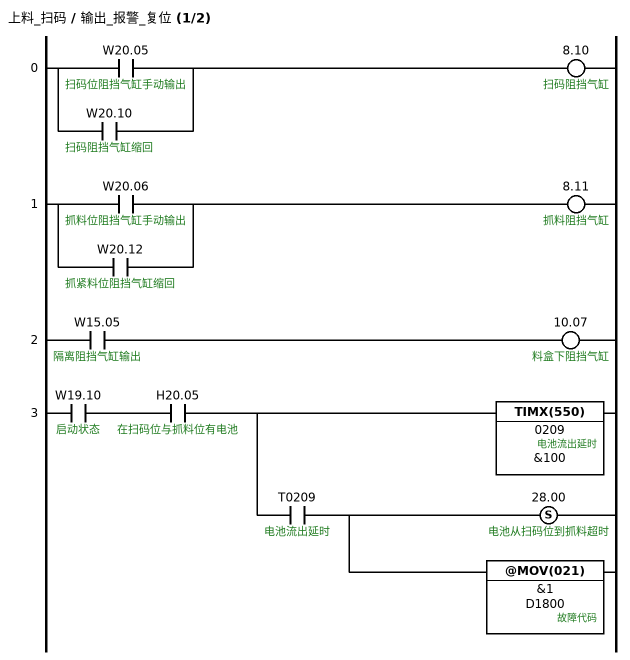
; [picture p72: 上料_扫码 / 输出_报警_复位, rungs 0-3]
; rung 0
LD W20.05  ; 扫码位阻挡气缸手动输出
OR W20.10  ; 扫码阻挡气缸缩回
OUT 8.10  ; 扫码阻挡气缸
; rung 1
LD W20.06  ; 抓料位阻挡气缸手动输出
OR W20.12  ; 抓紧料位阻挡气缸缩回
OUT 8.11  ; 抓料阻挡气缸
; rung 2
LD W15.05  ; 隔离阻挡气缸输出
OUT 10.07  ; 料盒下阻挡气缸
; rung 3
LD W19.10  ; 启动状态
AND H20.05  ; 在扫码位与抓料位有电池
TIMX(550) 0209 &100  ; 电池流出延时
AND T0209  ; 电池流出延时
SET 28.00  ; 电池从扫码位到抓料超时
@MOV(021) &1 D1800  ; 故障代码

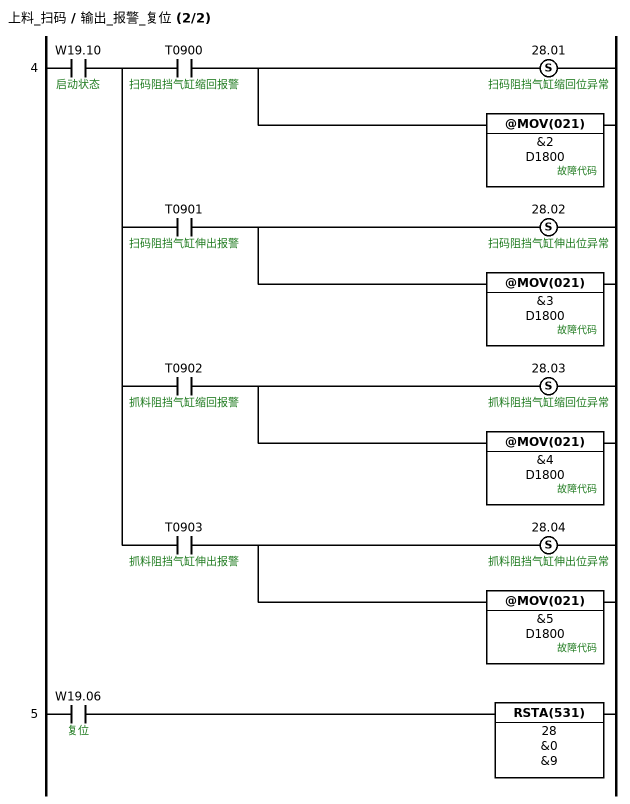
; rung 4
LD W19.10  ; 启动状态
OUT TR0
AND T0900  ; 扫码阻挡气缸缩回报警
SET 28.01  ; 扫码阻挡气缸缩回位异常
@MOV(021) &2 D1800  ; 故障代码
LD TR0
AND T0901  ; 扫码阻挡气缸伸出报警
SET 28.02  ; 扫码阻挡气缸伸出位异常
@MOV(021) &3 D1800  ; 故障代码
LD TR0
AND T0902  ; 抓料阻挡气缸缩回报警
SET 28.03  ; 抓料阻挡气缸缩回位异常
@MOV(021) &4 D1800  ; 故障代码
LD TR0
AND T0903  ; 抓料阻挡气缸伸出报警
SET 28.04  ; 抓料阻挡气缸伸出位异常
@MOV(021) &5 D1800  ; 故障代码
; rung 5
LD W19.06  ; 复位
RSTA(531) 28 &0 &9

### Section END
; rung 0
END(001)

## Program 上料机手 (cyclic task 2)

### Section 上料机械手手动

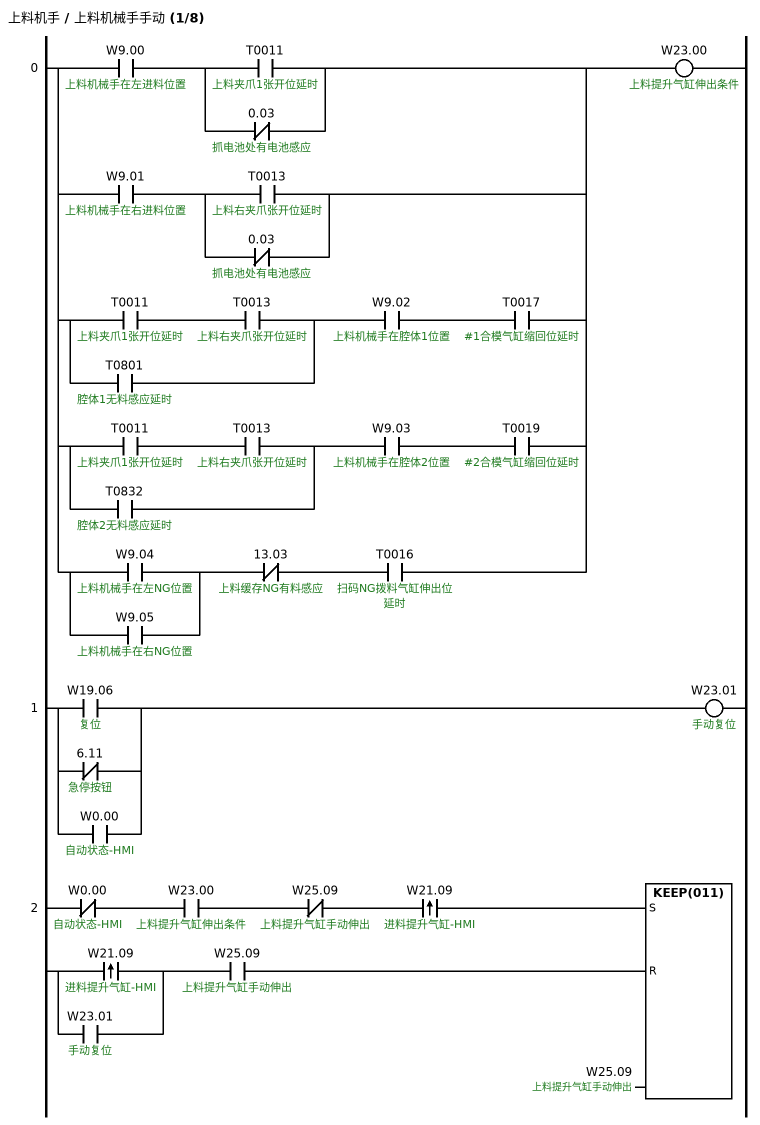
; rung 0
LD W9.00  ; 上料机械手在左进料位置
LD T0011  ; 上料夹爪1张开位延时
ORNOT 0.03  ; 抓电池处有电池感应
ANDLD
LD W9.01  ; 上料机械手在右进料位置
LD T0013  ; 上料右夹爪张开位延时
ORNOT 0.03  ; 抓电池处有电池感应
ANDLD
ORLD
LD T0011  ; 上料夹爪1张开位延时
AND T0013  ; 上料右夹爪张开位延时
OR T0801  ; 腔体1无料感应延时
AND W9.02  ; 上料机械手在腔体1位置
AND T0017  ; #1合模气缸缩回位延时
ORLD
LD T0011  ; 上料夹爪1张开位延时
AND T0013  ; 上料右夹爪张开位延时
OR T0832  ; 腔体2无料感应延时
AND W9.03  ; 上料机械手在腔体2位置
AND T0019  ; #2合模气缸缩回位延时
ORLD
LD W9.04  ; 上料机械手在左NG位置
OR W9.05  ; 上料机械手在右NG位置
ANDNOT 13.03  ; 上料缓存NG有料感应
AND T0016  ; 扫码NG拨料气缸伸出位延时
ORLD
OUT W23.00  ; 上料提升气缸伸出条件
; rung 1
LD W19.06  ; 复位
ORNOT 6.11  ; 急停按钮
OR W0.00  ; 自动状态-HMI
OUT W23.01  ; 手动复位
; rung 2
LDNOT W0.00  ; 自动状态-HMI
AND W23.00  ; 上料提升气缸伸出条件
ANDNOT W25.09  ; 上料提升气缸手动伸出
@AND W21.09  ; 进料提升气缸-HMI
@LD W21.09  ; 进料提升气缸-HMI
OR W23.01  ; 手动复位
AND W25.09  ; 上料提升气缸手动伸出
KEEP(011) W25.09  ; 上料提升气缸手动伸出

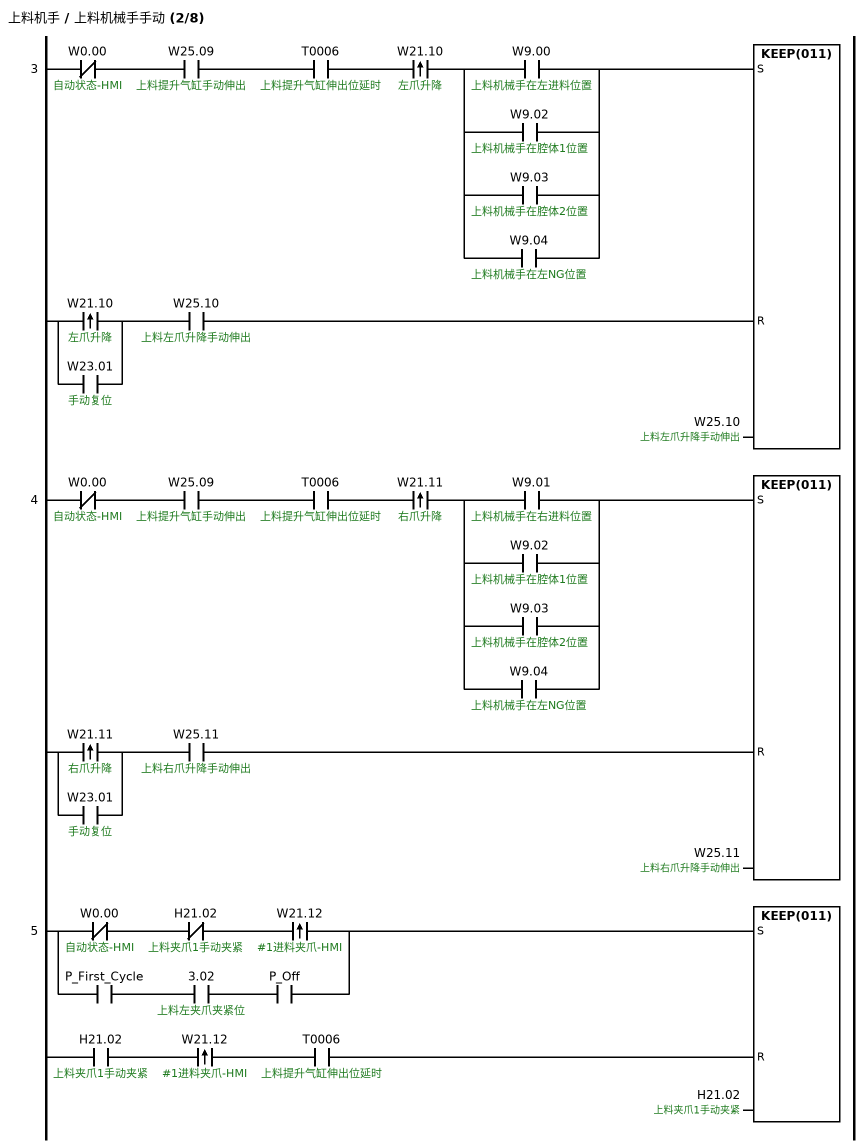
; rung 3
LDNOT W0.00  ; 自动状态-HMI
AND W25.09  ; 上料提升气缸手动伸出
AND T0006  ; 上料提升气缸伸出位延时
@AND W21.10  ; 左爪升降
LD W9.00  ; 上料机械手在左进料位置
OR W9.02  ; 上料机械手在腔体1位置
OR W9.03  ; 上料机械手在腔体2位置
OR W9.04  ; 上料机械手在左NG位置
ANDLD
@LD W21.10  ; 左爪升降
OR W23.01  ; 手动复位
AND W25.10  ; 上料左爪升降手动伸出
KEEP(011) W25.10  ; 上料左爪升降手动伸出
; rung 4
LDNOT W0.00  ; 自动状态-HMI
AND W25.09  ; 上料提升气缸手动伸出
AND T0006  ; 上料提升气缸伸出位延时
@AND W21.11  ; 右爪升降
LD W9.01  ; 上料机械手在右进料位置
OR W9.02  ; 上料机械手在腔体1位置
OR W9.03  ; 上料机械手在腔体2位置
OR W9.04  ; 上料机械手在左NG位置
ANDLD
@LD W21.11  ; 右爪升降
OR W23.01  ; 手动复位
AND W25.11  ; 上料右爪升降手动伸出
KEEP(011) W25.11  ; 上料右爪升降手动伸出
; rung 5
LDNOT W0.00  ; 自动状态-HMI
ANDNOT H21.02  ; 上料夹爪1手动夹紧
@AND W21.12  ; #1进料夹爪-HMI
LD P_First_Cycle
AND 3.02  ; 上料左夹爪夹紧位
AND P_Off
ORLD
LD H21.02  ; 上料夹爪1手动夹紧
@AND W21.12  ; #1进料夹爪-HMI
AND T0006  ; 上料提升气缸伸出位延时
KEEP(011) H21.02  ; 上料夹爪1手动夹紧

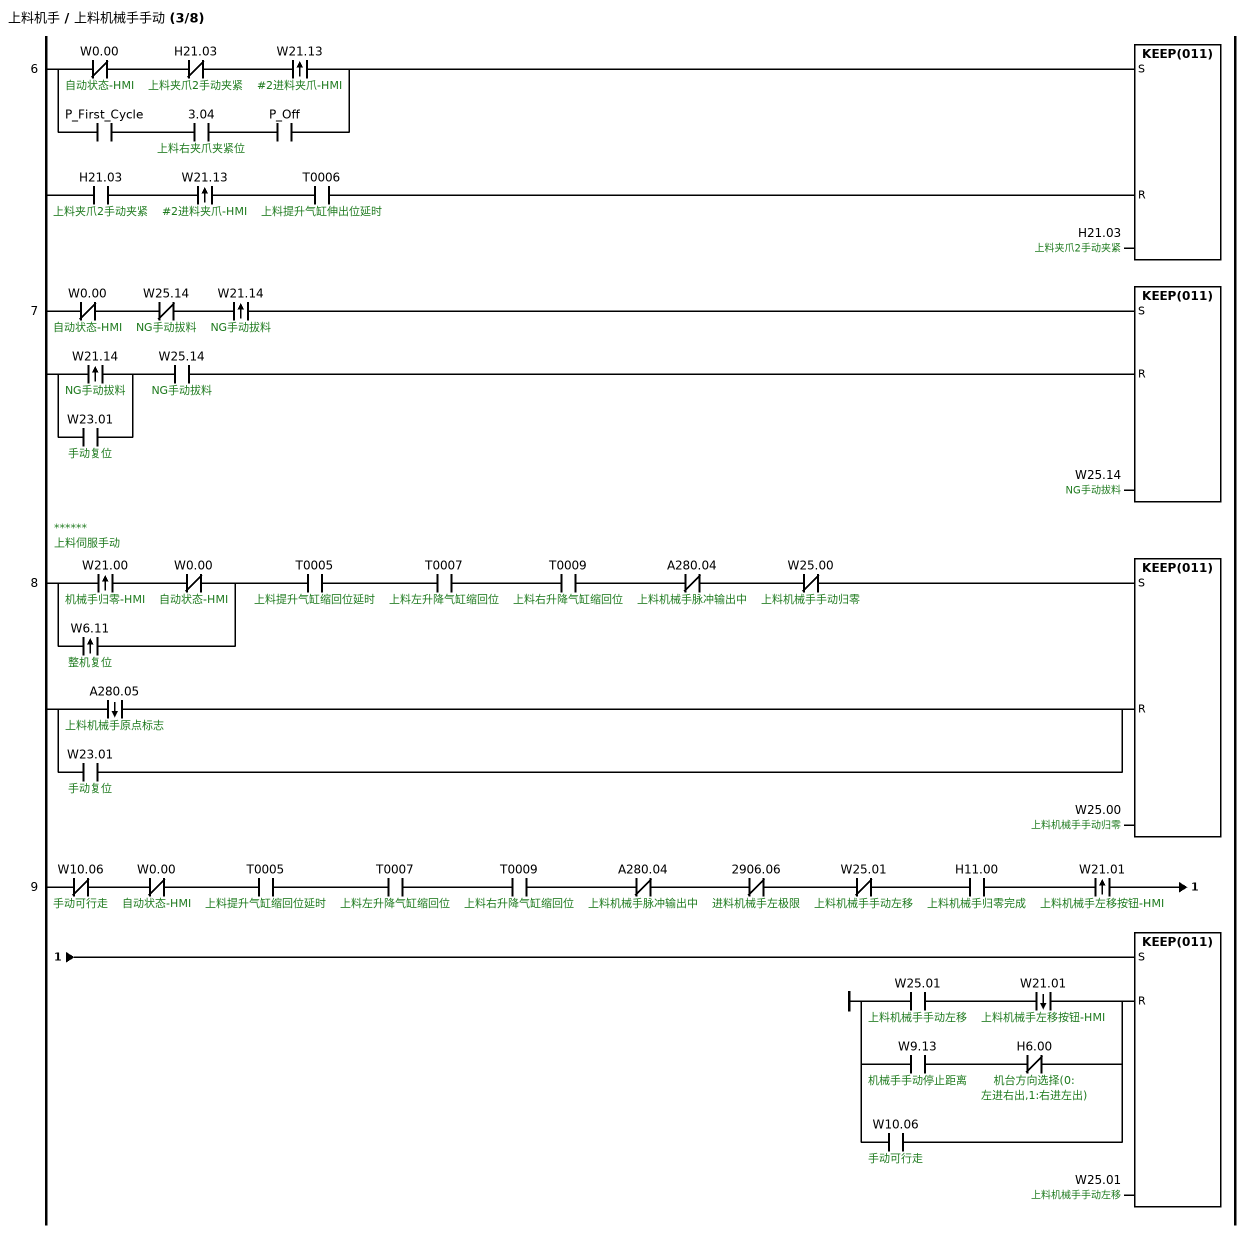
; rung 6
LDNOT W0.00  ; 自动状态-HMI
ANDNOT H21.03  ; 上料夹爪2手动夹紧
@AND W21.13  ; #2进料夹爪-HMI
LD P_First_Cycle
AND 3.04  ; 上料右夹爪夹紧位
AND P_Off
ORLD
LD H21.03  ; 上料夹爪2手动夹紧
@AND W21.13  ; #2进料夹爪-HMI
AND T0006  ; 上料提升气缸伸出位延时
KEEP(011) H21.03  ; 上料夹爪2手动夹紧
; rung 7
LDNOT W0.00  ; 自动状态-HMI
ANDNOT W25.14  ; NG手动拔料
@AND W21.14  ; NG手动拔料
@LD W21.14  ; NG手动拔料
OR W23.01  ; 手动复位
AND W25.14  ; NG手动拔料
KEEP(011) W25.14  ; NG手动拔料
; rung 8: ****** / 上料伺服手动
@LD W21.00  ; 机械手归零-HMI
ANDNOT W0.00  ; 自动状态-HMI
@OR W6.11  ; 整机复位
AND T0005  ; 上料提升气缸缩回位延时
AND T0007  ; 上料左升降气缸缩回位
AND T0009  ; 上料右升降气缸缩回位
ANDNOT A280.04  ; 上料机械手脉冲输出中
ANDNOT W25.00  ; 上料机械手手动归零
%LD A280.05  ; 上料机械手原点标志
OR W23.01  ; 手动复位
KEEP(011) W25.00  ; 上料机械手手动归零
; rung 9
LDNOT W10.06  ; 手动可行走
ANDNOT W0.00  ; 自动状态-HMI
AND T0005  ; 上料提升气缸缩回位延时
AND T0007  ; 上料左升降气缸缩回位
AND T0009  ; 上料右升降气缸缩回位
ANDNOT A280.04  ; 上料机械手脉冲输出中
ANDNOT 2906.06  ; 进料机械手左极限
ANDNOT W25.01  ; 上料机械手手动左移
AND H11.00  ; 上料机械手归零完成
@AND W21.01  ; 上料机械手左移按钮-HMI
LD W25.01  ; 上料机械手手动左移
%AND W21.01  ; 上料机械手左移按钮-HMI
LD W9.13  ; 机械手手动停止距离
ANDNOT H6.00  ; 机台方向选择(0:左进右出,1:右进左出)
ORLD
OR W10.06  ; 手动可行走
KEEP(011) W25.01  ; 上料机械手手动左移

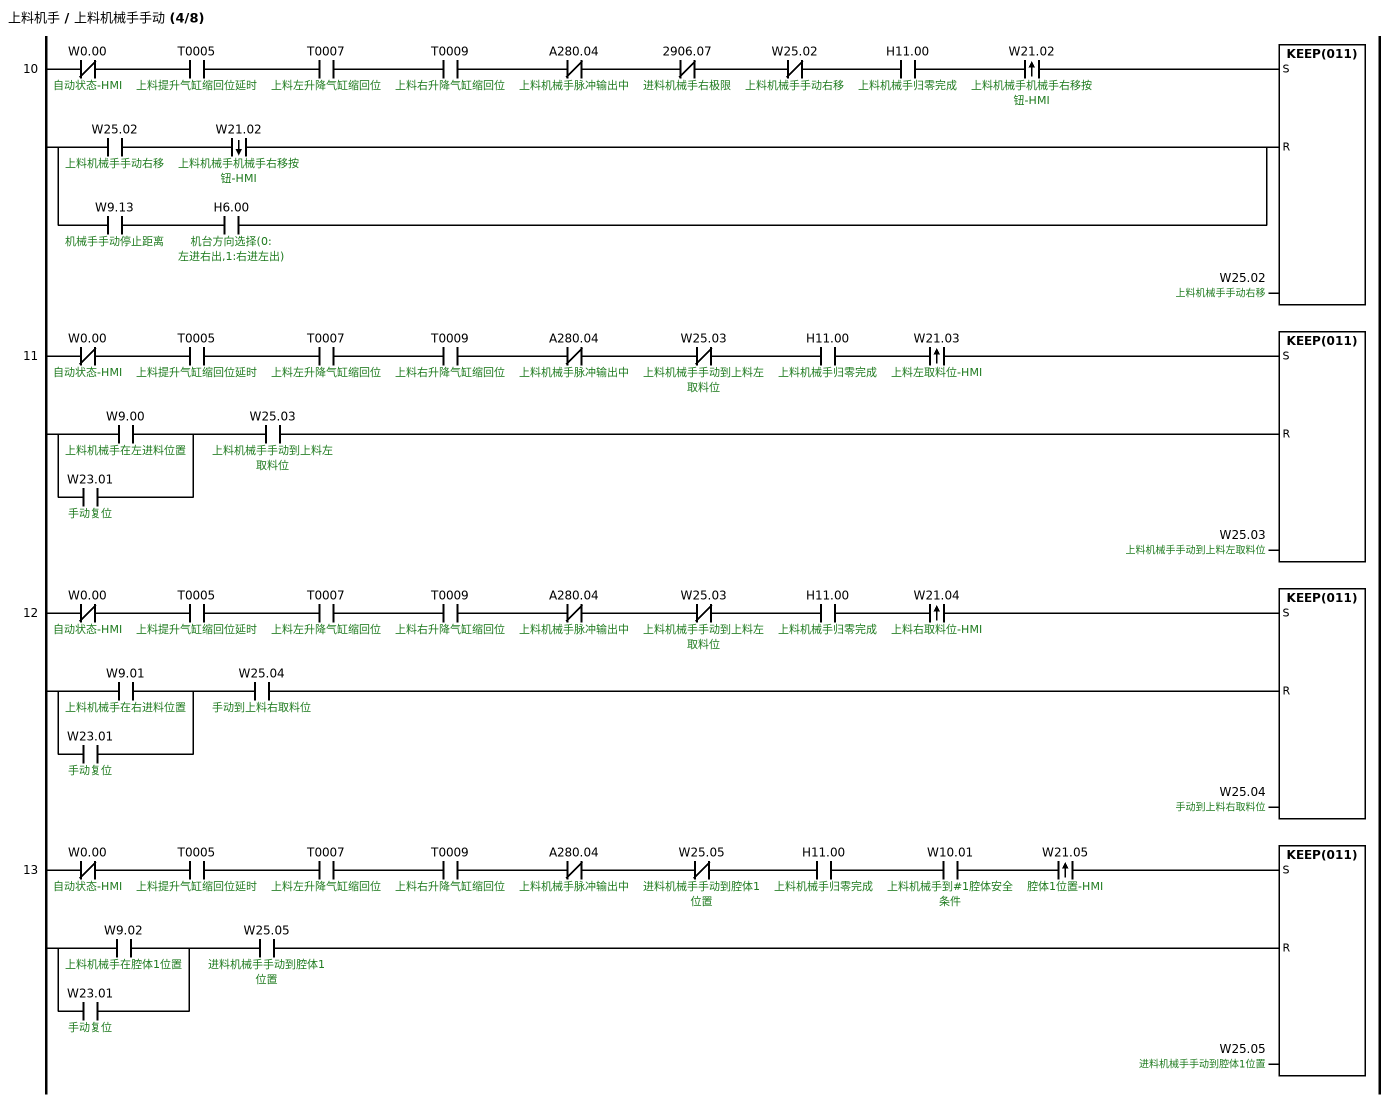
; rung 10
LDNOT W0.00  ; 自动状态-HMI
AND T0005  ; 上料提升气缸缩回位延时
AND T0007  ; 上料左升降气缸缩回位
AND T0009  ; 上料右升降气缸缩回位
ANDNOT A280.04  ; 上料机械手脉冲输出中
ANDNOT 2906.07  ; 进料机械手右极限
ANDNOT W25.02  ; 上料机械手手动右移
AND H11.00  ; 上料机械手归零完成
@AND W21.02  ; 上料机械手机械手右移按钮-HMI
LD W25.02  ; 上料机械手手动右移
%AND W21.02  ; 上料机械手机械手右移按钮-HMI
LD W9.13  ; 机械手手动停止距离
AND H6.00  ; 机台方向选择(0:左进右出,1:右进左出)
ORLD
KEEP(011) W25.02  ; 上料机械手手动右移
; rung 11
LDNOT W0.00  ; 自动状态-HMI
AND T0005  ; 上料提升气缸缩回位延时
AND T0007  ; 上料左升降气缸缩回位
AND T0009  ; 上料右升降气缸缩回位
ANDNOT A280.04  ; 上料机械手脉冲输出中
ANDNOT W25.03  ; 上料机械手手动到上料左取料位
AND H11.00  ; 上料机械手归零完成
@AND W21.03  ; 上料左取料位-HMI
LD W9.00  ; 上料机械手在左进料位置
OR W23.01  ; 手动复位
AND W25.03  ; 上料机械手手动到上料左取料位
KEEP(011) W25.03  ; 上料机械手手动到上料左取料位
; rung 12
LDNOT W0.00  ; 自动状态-HMI
AND T0005  ; 上料提升气缸缩回位延时
AND T0007  ; 上料左升降气缸缩回位
AND T0009  ; 上料右升降气缸缩回位
ANDNOT A280.04  ; 上料机械手脉冲输出中
ANDNOT W25.03  ; 上料机械手手动到上料左取料位
AND H11.00  ; 上料机械手归零完成
@AND W21.04  ; 上料右取料位-HMI
LD W9.01  ; 上料机械手在右进料位置
OR W23.01  ; 手动复位
AND W25.04  ; 手动到上料右取料位
KEEP(011) W25.04  ; 手动到上料右取料位
; rung 13
LDNOT W0.00  ; 自动状态-HMI
AND T0005  ; 上料提升气缸缩回位延时
AND T0007  ; 上料左升降气缸缩回位
AND T0009  ; 上料右升降气缸缩回位
ANDNOT A280.04  ; 上料机械手脉冲输出中
ANDNOT W25.05  ; 进料机械手手动到腔体1位置
AND H11.00  ; 上料机械手归零完成
AND W10.01  ; 上料机械手到#1腔体安全条件
@AND W21.05  ; 腔体1位置-HMI
LD W9.02  ; 上料机械手在腔体1位置
OR W23.01  ; 手动复位
AND W25.05  ; 进料机械手手动到腔体1位置
KEEP(011) W25.05  ; 进料机械手手动到腔体1位置

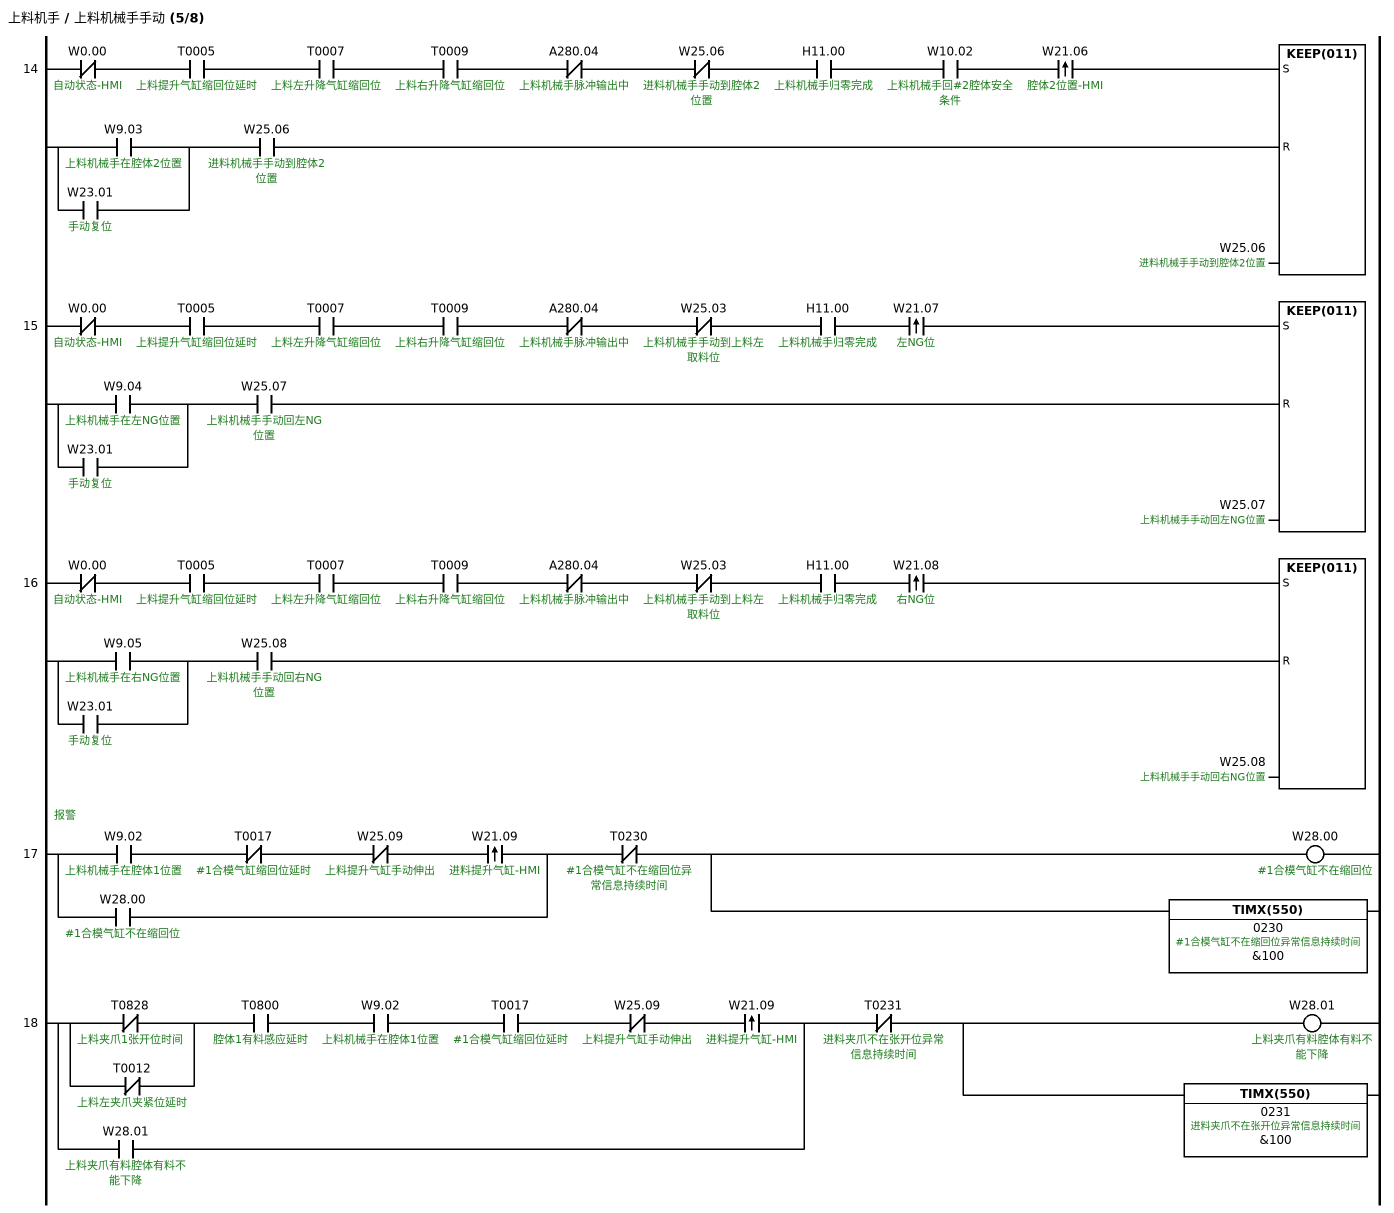
; rung 14
LDNOT W0.00  ; 自动状态-HMI
AND T0005  ; 上料提升气缸缩回位延时
AND T0007  ; 上料左升降气缸缩回位
AND T0009  ; 上料右升降气缸缩回位
ANDNOT A280.04  ; 上料机械手脉冲输出中
ANDNOT W25.06  ; 进料机械手手动到腔体2位置
AND H11.00  ; 上料机械手归零完成
AND W10.02  ; 上料机械手回#2腔体安全条件
@AND W21.06  ; 腔体2位置-HMI
LD W9.03  ; 上料机械手在腔体2位置
OR W23.01  ; 手动复位
AND W25.06  ; 进料机械手手动到腔体2位置
KEEP(011) W25.06  ; 进料机械手手动到腔体2位置
; rung 15
LDNOT W0.00  ; 自动状态-HMI
AND T0005  ; 上料提升气缸缩回位延时
AND T0007  ; 上料左升降气缸缩回位
AND T0009  ; 上料右升降气缸缩回位
ANDNOT A280.04  ; 上料机械手脉冲输出中
ANDNOT W25.03  ; 上料机械手手动到上料左取料位
AND H11.00  ; 上料机械手归零完成
@AND W21.07  ; 左NG位
LD W9.04  ; 上料机械手在左NG位置
OR W23.01  ; 手动复位
AND W25.07  ; 上料机械手手动回左NG位置
KEEP(011) W25.07  ; 上料机械手手动回左NG位置
; rung 16
LDNOT W0.00  ; 自动状态-HMI
AND T0005  ; 上料提升气缸缩回位延时
AND T0007  ; 上料左升降气缸缩回位
AND T0009  ; 上料右升降气缸缩回位
ANDNOT A280.04  ; 上料机械手脉冲输出中
ANDNOT W25.03  ; 上料机械手手动到上料左取料位
AND H11.00  ; 上料机械手归零完成
@AND W21.08  ; 右NG位
LD W9.05  ; 上料机械手在右NG位置
OR W23.01  ; 手动复位
AND W25.08  ; 上料机械手手动回右NG位置
KEEP(011) W25.08  ; 上料机械手手动回右NG位置
; rung 17: 报警
LD W9.02  ; 上料机械手在腔体1位置
ANDNOT T0017  ; #1合模气缸缩回位延时
ANDNOT W25.09  ; 上料提升气缸手动伸出
@AND W21.09  ; 进料提升气缸-HMI
OR W28.00  ; #1合模气缸不在缩回位
ANDNOT T0230  ; #1合模气缸不在缩回位异常信息持续时间
OUT W28.00  ; #1合模气缸不在缩回位
TIMX(550) 0230 &100  ; #1合模气缸不在缩回位异常信息持续时间
; rung 18
LDNOT T0828  ; 上料夹爪1张开位时间
ORNOT T0012  ; 上料左夹爪夹紧位延时
AND T0800  ; 腔体1有料感应延时
AND W9.02  ; 上料机械手在腔体1位置
AND T0017  ; #1合模气缸缩回位延时
ANDNOT W25.09  ; 上料提升气缸手动伸出
@AND W21.09  ; 进料提升气缸-HMI
OR W28.01  ; 上料夹爪有料腔体有料不能下降
ANDNOT T0231  ; 进料夹爪不在张开位异常信息持续时间
OUT W28.01  ; 上料夹爪有料腔体有料不能下降
TIMX(550) 0231 &100  ; 进料夹爪不在张开位异常信息持续时间

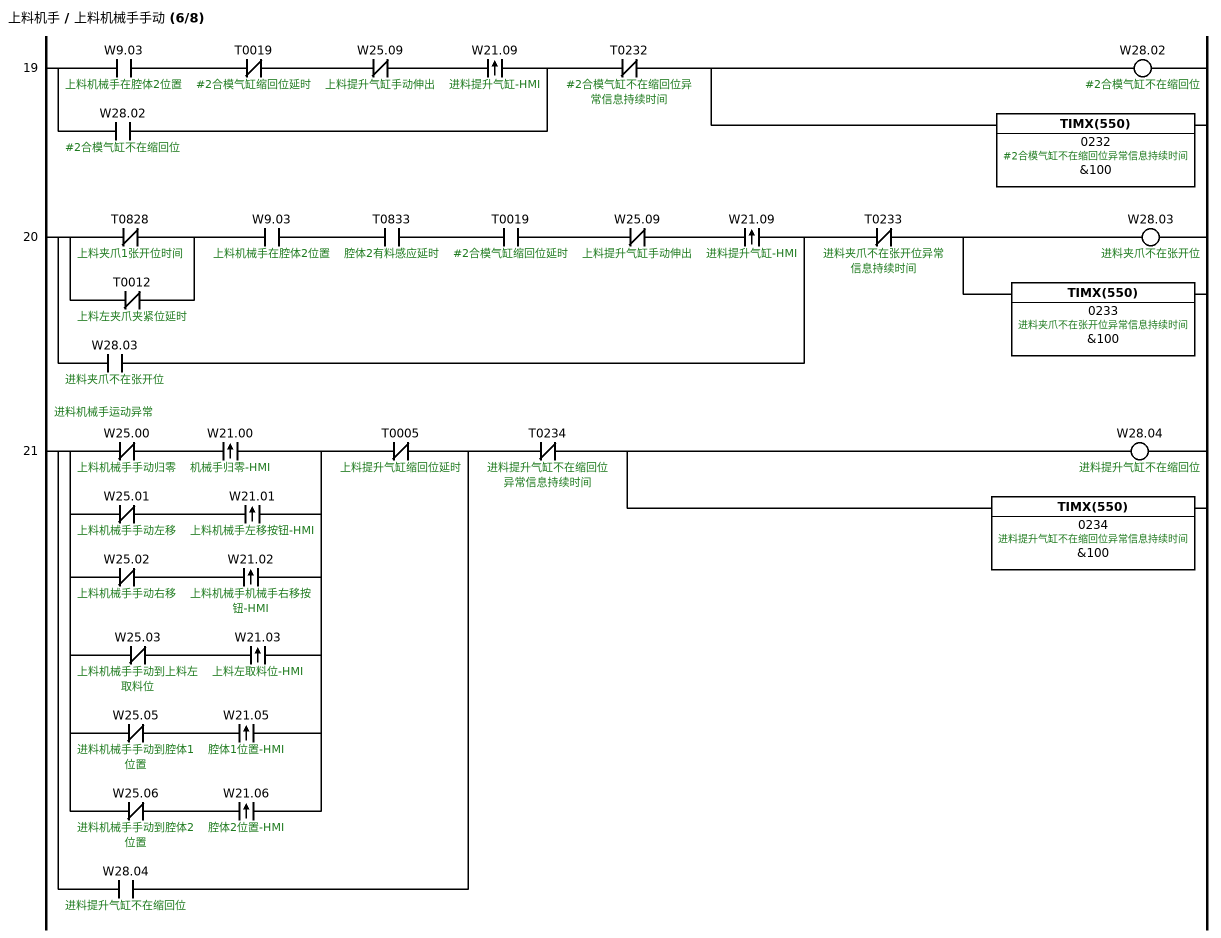
; rung 19
LD W9.03  ; 上料机械手在腔体2位置
ANDNOT T0019  ; #2合模气缸缩回位延时
ANDNOT W25.09  ; 上料提升气缸手动伸出
@AND W21.09  ; 进料提升气缸-HMI
OR W28.02  ; #2合模气缸不在缩回位
ANDNOT T0232  ; #2合模气缸不在缩回位异常信息持续时间
OUT W28.02  ; #2合模气缸不在缩回位
TIMX(550) 0232 &100  ; #2合模气缸不在缩回位异常信息持续时间
; rung 20
LDNOT T0828  ; 上料夹爪1张开位时间
ORNOT T0012  ; 上料左夹爪夹紧位延时
AND W9.03  ; 上料机械手在腔体2位置
AND T0833  ; 腔体2有料感应延时
AND T0019  ; #2合模气缸缩回位延时
ANDNOT W25.09  ; 上料提升气缸手动伸出
@AND W21.09  ; 进料提升气缸-HMI
OR W28.03  ; 进料夹爪不在张开位
ANDNOT T0233  ; 进料夹爪不在张开位异常信息持续时间
OUT W28.03  ; 进料夹爪不在张开位
TIMX(550) 0233 &100  ; 进料夹爪不在张开位异常信息持续时间
; rung 21: 进料机械手运动异常
LDNOT W25.00  ; 上料机械手手动归零
@AND W21.00  ; 机械手归零-HMI
LDNOT W25.01  ; 上料机械手手动左移
@AND W21.01  ; 上料机械手左移按钮-HMI
ORLD
LDNOT W25.02  ; 上料机械手手动右移
@AND W21.02  ; 上料机械手机械手右移按钮-HMI
ORLD
LDNOT W25.03  ; 上料机械手手动到上料左取料位
@AND W21.03  ; 上料左取料位-HMI
ORLD
LDNOT W25.05  ; 进料机械手手动到腔体1位置
@AND W21.05  ; 腔体1位置-HMI
ORLD
LDNOT W25.06  ; 进料机械手手动到腔体2位置
@AND W21.06  ; 腔体2位置-HMI
ORLD
ANDNOT T0005  ; 上料提升气缸缩回位延时
OR W28.04  ; 进料提升气缸不在缩回位
ANDNOT T0234  ; 进料提升气缸不在缩回位异常信息持续时间
OUT W28.04  ; 进料提升气缸不在缩回位
TIMX(550) 0234 &100  ; 进料提升气缸不在缩回位异常信息持续时间

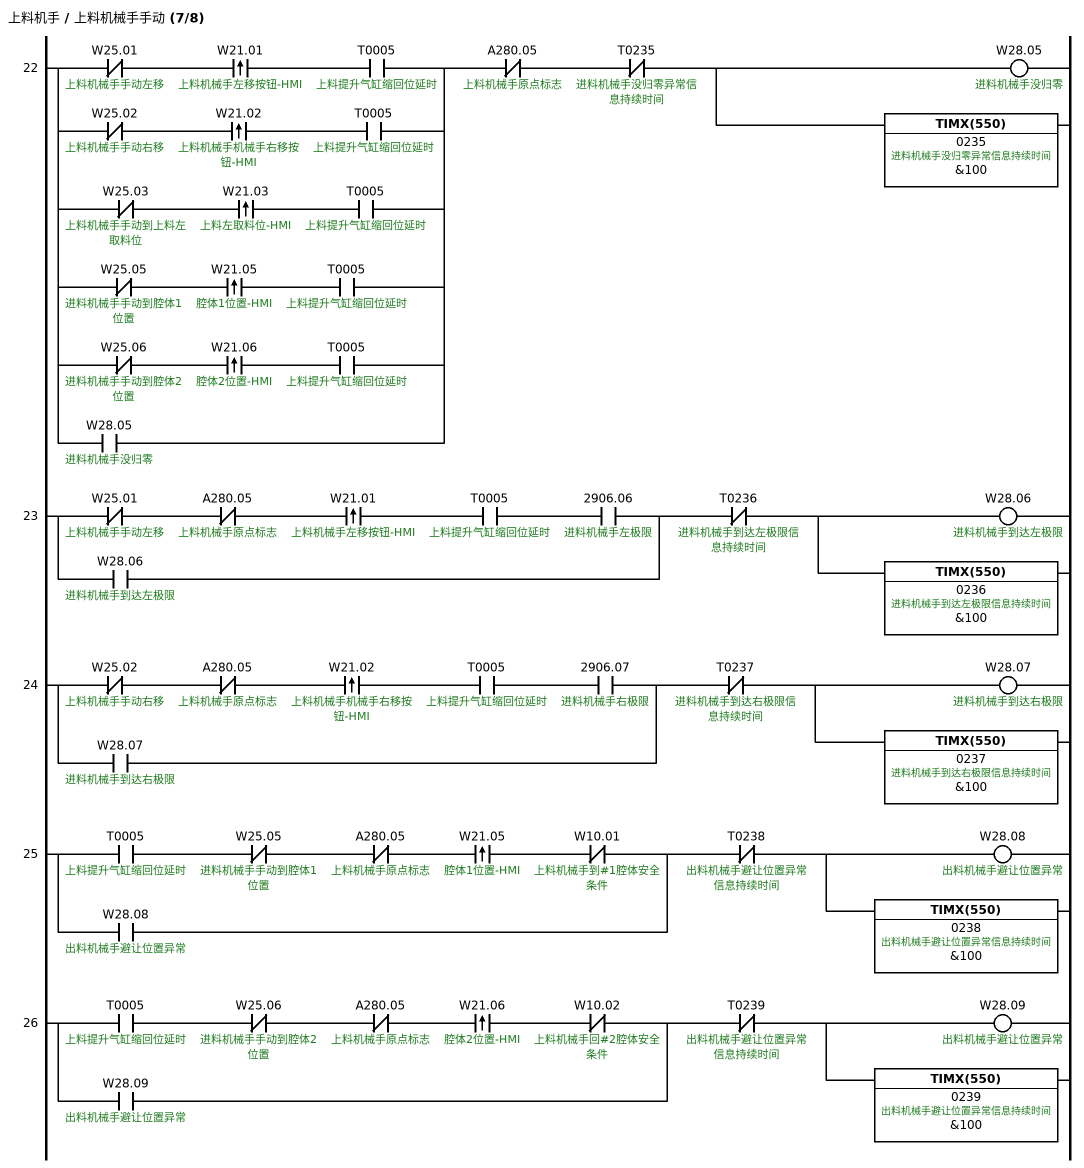
; rung 22
LDNOT W25.01  ; 上料机械手手动左移
@AND W21.01  ; 上料机械手左移按钮-HMI
AND T0005  ; 上料提升气缸缩回位延时
LDNOT W25.02  ; 上料机械手手动右移
@AND W21.02  ; 上料机械手机械手右移按钮-HMI
AND T0005  ; 上料提升气缸缩回位延时
ORLD
LDNOT W25.03  ; 上料机械手手动到上料左取料位
@AND W21.03  ; 上料左取料位-HMI
AND T0005  ; 上料提升气缸缩回位延时
ORLD
LDNOT W25.05  ; 进料机械手手动到腔体1位置
@AND W21.05  ; 腔体1位置-HMI
AND T0005  ; 上料提升气缸缩回位延时
ORLD
LDNOT W25.06  ; 进料机械手手动到腔体2位置
@AND W21.06  ; 腔体2位置-HMI
AND T0005  ; 上料提升气缸缩回位延时
ORLD
OR W28.05  ; 进料机械手没归零
ANDNOT A280.05  ; 上料机械手原点标志
ANDNOT T0235  ; 进料机械手没归零异常信息持续时间
OUT W28.05  ; 进料机械手没归零
TIMX(550) 0235 &100  ; 进料机械手没归零异常信息持续时间
; rung 23
LDNOT W25.01  ; 上料机械手手动左移
ANDNOT A280.05  ; 上料机械手原点标志
@AND W21.01  ; 上料机械手左移按钮-HMI
AND T0005  ; 上料提升气缸缩回位延时
AND 2906.06  ; 进料机械手左极限
OR W28.06  ; 进料机械手到达左极限
ANDNOT T0236  ; 进料机械手到达左极限信息持续时间
OUT W28.06  ; 进料机械手到达左极限
TIMX(550) 0236 &100  ; 进料机械手到达左极限信息持续时间
; rung 24
LDNOT W25.02  ; 上料机械手手动右移
ANDNOT A280.05  ; 上料机械手原点标志
@AND W21.02  ; 上料机械手机械手右移按钮-HMI
AND T0005  ; 上料提升气缸缩回位延时
AND 2906.07  ; 进料机械手右极限
OR W28.07  ; 进料机械手到达右极限
ANDNOT T0237  ; 进料机械手到达右极限信息持续时间
OUT W28.07  ; 进料机械手到达右极限
TIMX(550) 0237 &100  ; 进料机械手到达右极限信息持续时间
; rung 25
LD T0005  ; 上料提升气缸缩回位延时
ANDNOT W25.05  ; 进料机械手手动到腔体1位置
ANDNOT A280.05  ; 上料机械手原点标志
@AND W21.05  ; 腔体1位置-HMI
ANDNOT W10.01  ; 上料机械手到#1腔体安全条件
OR W28.08  ; 出料机械手避让位置异常
ANDNOT T0238  ; 出料机械手避让位置异常信息持续时间
OUT W28.08  ; 出料机械手避让位置异常
TIMX(550) 0238 &100  ; 出料机械手避让位置异常信息持续时间
; rung 26
LD T0005  ; 上料提升气缸缩回位延时
ANDNOT W25.06  ; 进料机械手手动到腔体2位置
ANDNOT A280.05  ; 上料机械手原点标志
@AND W21.06  ; 腔体2位置-HMI
ANDNOT W10.02  ; 上料机械手回#2腔体安全条件
OR W28.09  ; 出料机械手避让位置异常
ANDNOT T0239  ; 出料机械手避让位置异常信息持续时间
OUT W28.09  ; 出料机械手避让位置异常
TIMX(550) 0239 &100  ; 出料机械手避让位置异常信息持续时间

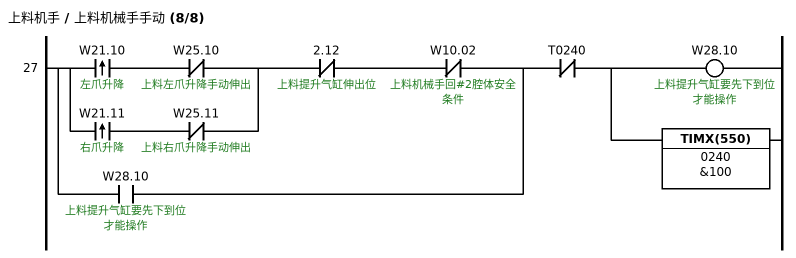
; rung 27
@LD W21.10  ; 左爪升降
ANDNOT W25.10  ; 上料左爪升降手动伸出
@LD W21.11  ; 右爪升降
ANDNOT W25.11  ; 上料右爪升降手动伸出
ORLD
ANDNOT 2.12  ; 上料提升气缸伸出位
ANDNOT W10.02  ; 上料机械手回#2腔体安全条件
OR W28.10  ; 上料提升气缸要先下到位才能操作
ANDNOT T0240
OUT W28.10  ; 上料提升气缸要先下到位才能操作
TIMX(550) 0240 &100

### Section 上料机械手自动

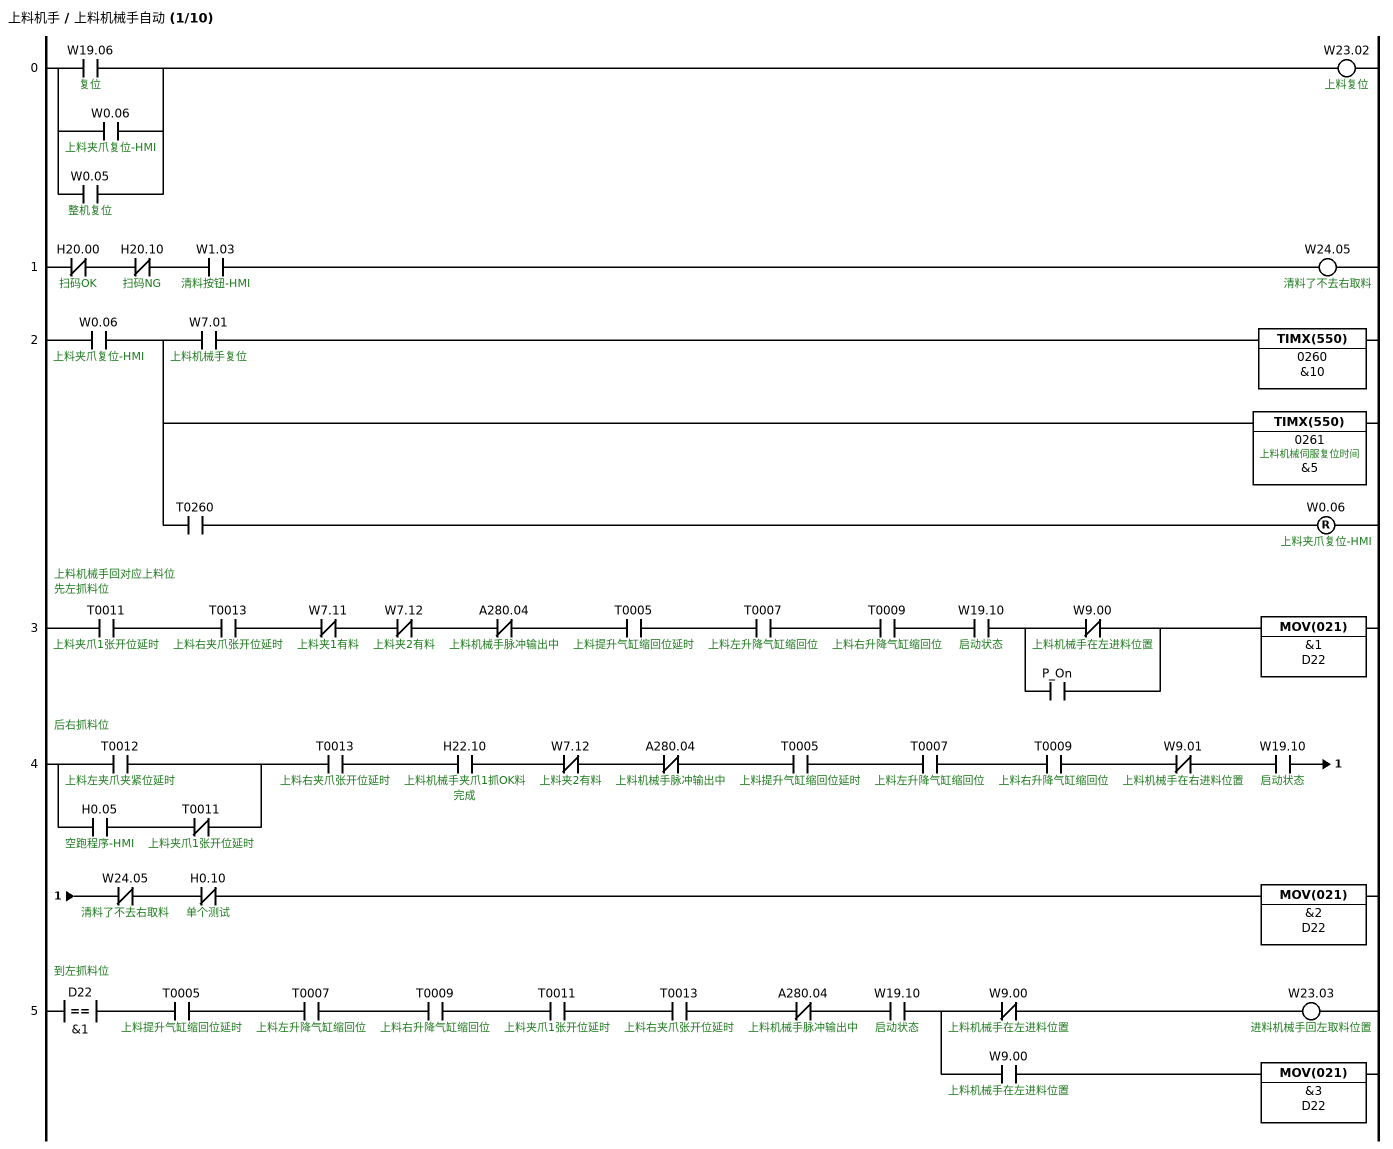
; rung 0
LD W19.06  ; 复位
OR W0.06  ; 上料夹爪复位-HMI
OR W0.05  ; 整机复位
OUT W23.02  ; 上料复位
; rung 1
LDNOT H20.00  ; 扫码OK
ANDNOT H20.10  ; 扫码NG
AND W1.03  ; 清料按钮-HMI
OUT W24.05  ; 清料了不去右取料
; rung 2
LD W0.06  ; 上料夹爪复位-HMI
OUT TR0
AND W7.01  ; 上料机械手复位
TIMX(550) 0260 &10
LD TR0
TIMX(550) 0261 &5  ; 上料机械伺服复位时间
AND T0260
RSET W0.06  ; 上料夹爪复位-HMI
; rung 3: 上料机械手回对应上料位 / 先左抓料位
LD T0011  ; 上料夹爪1张开位延时
AND T0013  ; 上料右夹爪张开位延时
ANDNOT W7.11  ; 上料夹1有料
ANDNOT W7.12  ; 上料夹2有料
ANDNOT A280.04  ; 上料机械手脉冲输出中
AND T0005  ; 上料提升气缸缩回位延时
AND T0007  ; 上料左升降气缸缩回位
AND T0009  ; 上料右升降气缸缩回位
AND W19.10  ; 启动状态
LDNOT W9.00  ; 上料机械手在左进料位置
OR P_On
ANDLD
MOV(021) &1 D22
; rung 4: 后右抓料位
LD T0012  ; 上料左夹爪夹紧位延时
LD H0.05  ; 空跑程序-HMI
ANDNOT T0011  ; 上料夹爪1张开位延时
ORLD
AND T0013  ; 上料右夹爪张开位延时
AND H22.10  ; 上料机械手夹爪1抓OK料完成
ANDNOT W7.12  ; 上料夹2有料
ANDNOT A280.04  ; 上料机械手脉冲输出中
AND T0005  ; 上料提升气缸缩回位延时
AND T0007  ; 上料左升降气缸缩回位
AND T0009  ; 上料右升降气缸缩回位
ANDNOT W9.01  ; 上料机械手在右进料位置
AND W19.10  ; 启动状态
ANDNOT W24.05  ; 清料了不去右取料
ANDNOT H0.10  ; 单个测试
MOV(021) &2 D22
; rung 5: 到左抓料位
LD=(300) D22 &1
AND T0005  ; 上料提升气缸缩回位延时
AND T0007  ; 上料左升降气缸缩回位
AND T0009  ; 上料右升降气缸缩回位
AND T0011  ; 上料夹爪1张开位延时
AND T0013  ; 上料右夹爪张开位延时
ANDNOT A280.04  ; 上料机械手脉冲输出中
AND W19.10  ; 启动状态
OUT TR0
ANDNOT W9.00  ; 上料机械手在左进料位置
OUT W23.03  ; 进料机械手回左取料位置
LD TR0
AND W9.00  ; 上料机械手在左进料位置
MOV(021) &3 D22

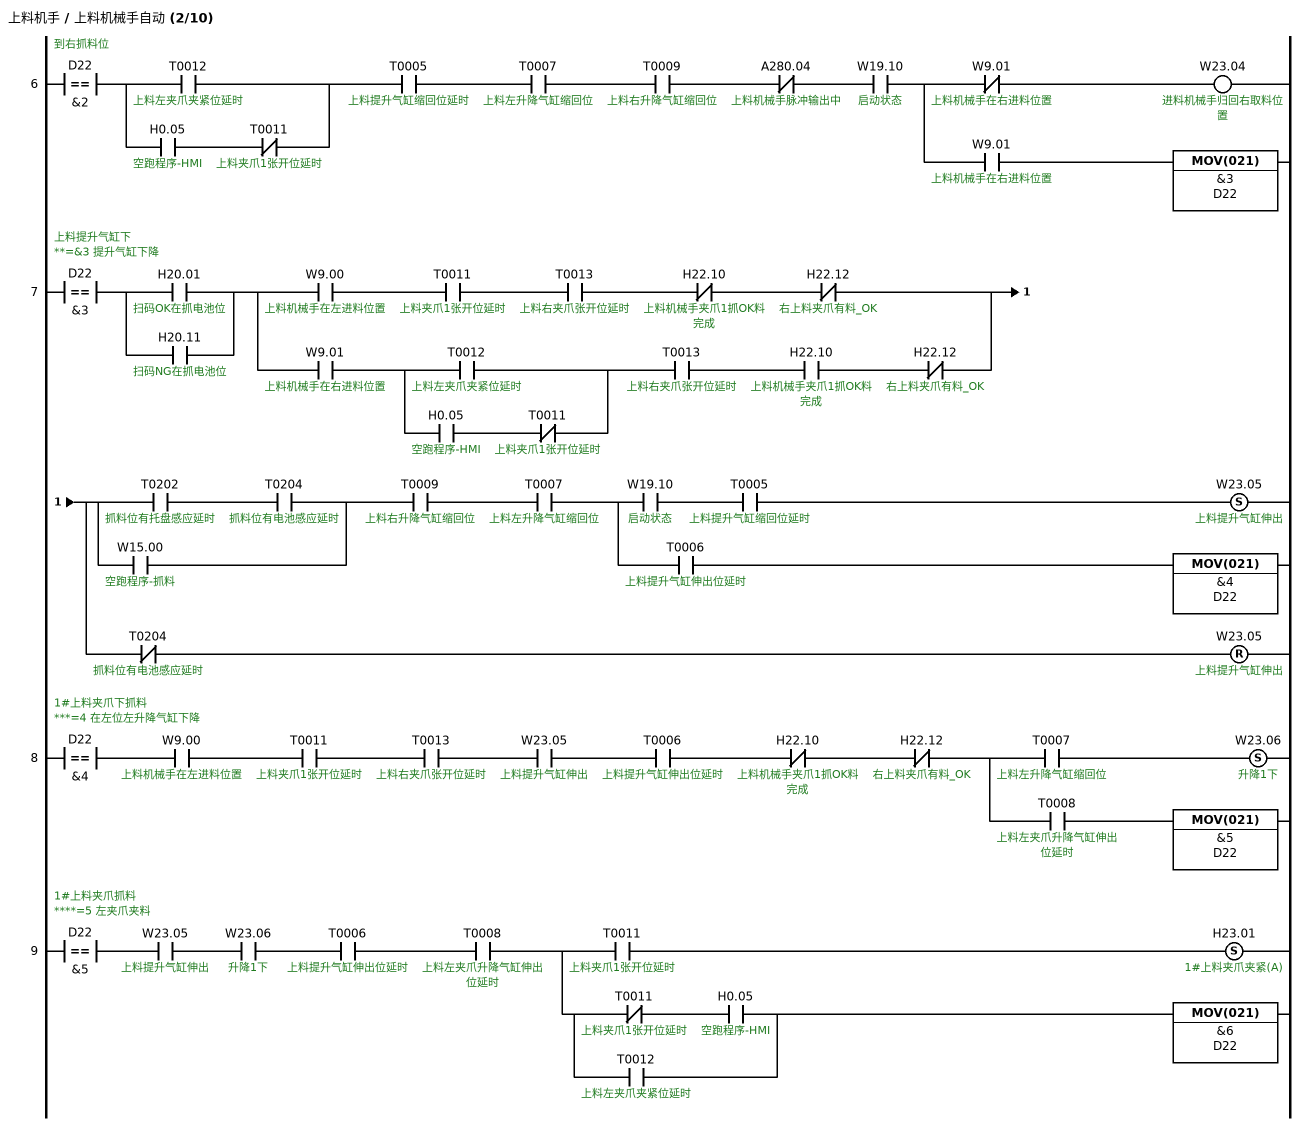
; rung 6: 到右抓料位
LD=(300) D22 &2
LD T0012  ; 上料左夹爪夹紧位延时
LD H0.05  ; 空跑程序-HMI
ANDNOT T0011  ; 上料夹爪1张开位延时
ORLD
ANDLD
AND T0005  ; 上料提升气缸缩回位延时
AND T0007  ; 上料左升降气缸缩回位
AND T0009  ; 上料右升降气缸缩回位
ANDNOT A280.04  ; 上料机械手脉冲输出中
AND W19.10  ; 启动状态
OUT TR0
ANDNOT W9.01  ; 上料机械手在右进料位置
OUT W23.04  ; 进料机械手归回右取料位置
LD TR0
AND W9.01  ; 上料机械手在右进料位置
MOV(021) &3 D22
; rung 7: 上料提升气缸下 / **=&3 提升气缸下降
LD=(300) D22 &3
LD H20.01  ; 扫码OK在抓电池位
OR H20.11  ; 扫码NG在抓电池位
ANDLD
LD W9.00  ; 上料机械手在左进料位置
AND T0011  ; 上料夹爪1张开位延时
AND T0013  ; 上料右夹爪张开位延时
ANDNOT H22.10  ; 上料机械手夹爪1抓OK料完成
ANDNOT H22.12  ; 右上料夹爪有料_OK
LD W9.01  ; 上料机械手在右进料位置
LD T0012  ; 上料左夹爪夹紧位延时
LD H0.05  ; 空跑程序-HMI
ANDNOT T0011  ; 上料夹爪1张开位延时
ORLD
ANDLD
AND T0013  ; 上料右夹爪张开位延时
AND H22.10  ; 上料机械手夹爪1抓OK料完成
ANDNOT H22.12  ; 右上料夹爪有料_OK
ORLD
ANDLD
OUT TR0
LD T0202  ; 抓料位有托盘感应延时
AND T0204  ; 抓料位有电池感应延时
OR W15.00  ; 空跑程序-抓料
ANDLD
AND T0009  ; 上料右升降气缸缩回位
AND T0007  ; 上料左升降气缸缩回位
OUT TR1
AND W19.10  ; 启动状态
AND T0005  ; 上料提升气缸缩回位延时
SET W23.05  ; 上料提升气缸伸出
LD TR1
AND T0006  ; 上料提升气缸伸出位延时
MOV(021) &4 D22
LD TR0
ANDNOT T0204  ; 抓料位有电池感应延时
RSET W23.05  ; 上料提升气缸伸出
; rung 8: 1#上料夹爪下抓料 / ***=4 在左位左升降气缸下降
LD=(300) D22 &4
AND W9.00  ; 上料机械手在左进料位置
AND T0011  ; 上料夹爪1张开位延时
AND T0013  ; 上料右夹爪张开位延时
AND W23.05  ; 上料提升气缸伸出
AND T0006  ; 上料提升气缸伸出位延时
ANDNOT H22.10  ; 上料机械手夹爪1抓OK料完成
ANDNOT H22.12  ; 右上料夹爪有料_OK
OUT TR0
AND T0007  ; 上料左升降气缸缩回位
SET W23.06  ; 升降1下
LD TR0
AND T0008  ; 上料左夹爪升降气缸伸出位延时
MOV(021) &5 D22
; rung 9: 1#上料夹爪抓料 / ****=5 左夹爪夹料
LD=(300) D22 &5
AND W23.05  ; 上料提升气缸伸出
AND W23.06  ; 升降1下
AND T0006  ; 上料提升气缸伸出位延时
AND T0008  ; 上料左夹爪升降气缸伸出位延时
OUT TR0
AND T0011  ; 上料夹爪1张开位延时
SET H23.01  ; 1#上料夹爪夹紧(A)
LD TR0
LDNOT T0011  ; 上料夹爪1张开位延时
AND H0.05  ; 空跑程序-HMI
OR T0012  ; 上料左夹爪夹紧位延时
ANDLD
MOV(021) &6 D22

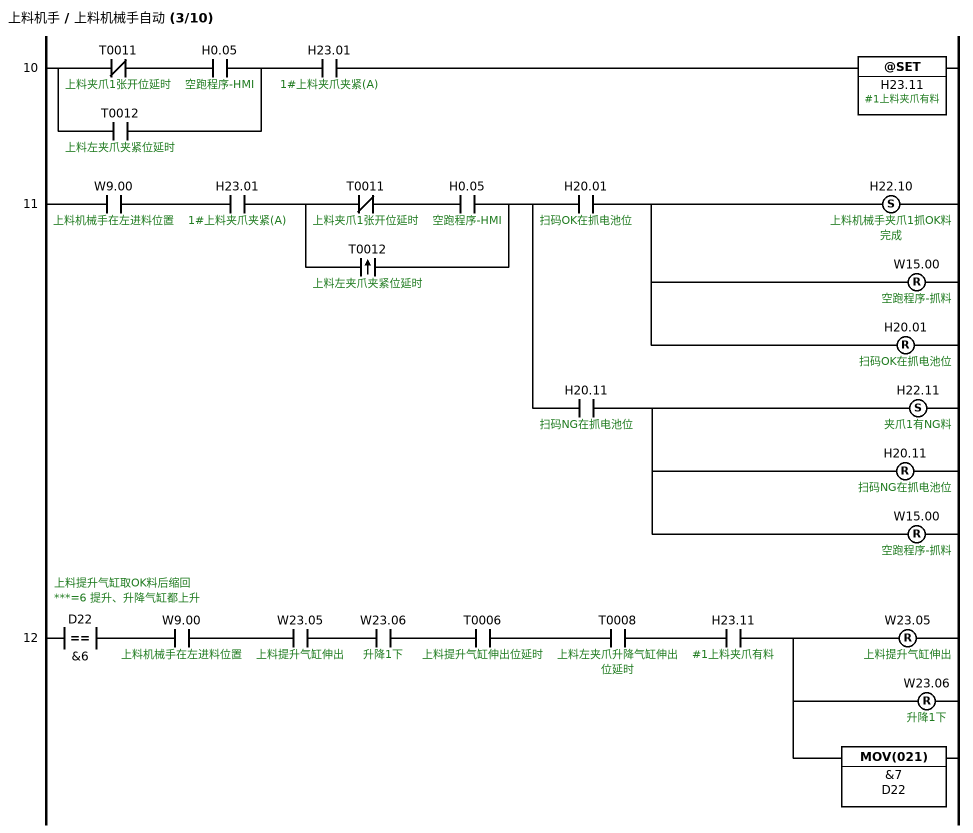
; rung 10
LDNOT T0011  ; 上料夹爪1张开位延时
AND H0.05  ; 空跑程序-HMI
OR T0012  ; 上料左夹爪夹紧位延时
AND H23.01  ; 1#上料夹爪夹紧(A)
@SET H23.11  ; #1上料夹爪有料
; rung 11
LD W9.00  ; 上料机械手在左进料位置
AND H23.01  ; 1#上料夹爪夹紧(A)
LDNOT T0011  ; 上料夹爪1张开位延时
AND H0.05  ; 空跑程序-HMI
@OR T0012  ; 上料左夹爪夹紧位延时
ANDLD
OUT TR0
AND H20.01  ; 扫码OK在抓电池位
SET H22.10  ; 上料机械手夹爪1抓OK料完成
RSET W15.00  ; 空跑程序-抓料
RSET H20.01  ; 扫码OK在抓电池位
LD TR0
AND H20.11  ; 扫码NG在抓电池位
SET H22.11  ; 夹爪1有NG料
RSET H20.11  ; 扫码NG在抓电池位
RSET W15.00  ; 空跑程序-抓料
; rung 12: 上料提升气缸取OK料后缩回 / ***=6 提升、升降气缸都上升
LD=(300) D22 &6
AND W9.00  ; 上料机械手在左进料位置
AND W23.05  ; 上料提升气缸伸出
AND W23.06  ; 升降1下
AND T0006  ; 上料提升气缸伸出位延时
AND T0008  ; 上料左夹爪升降气缸伸出位延时
AND H23.11  ; #1上料夹爪有料
RSET W23.05  ; 上料提升气缸伸出
RSET W23.06  ; 升降1下
MOV(021) &7 D22

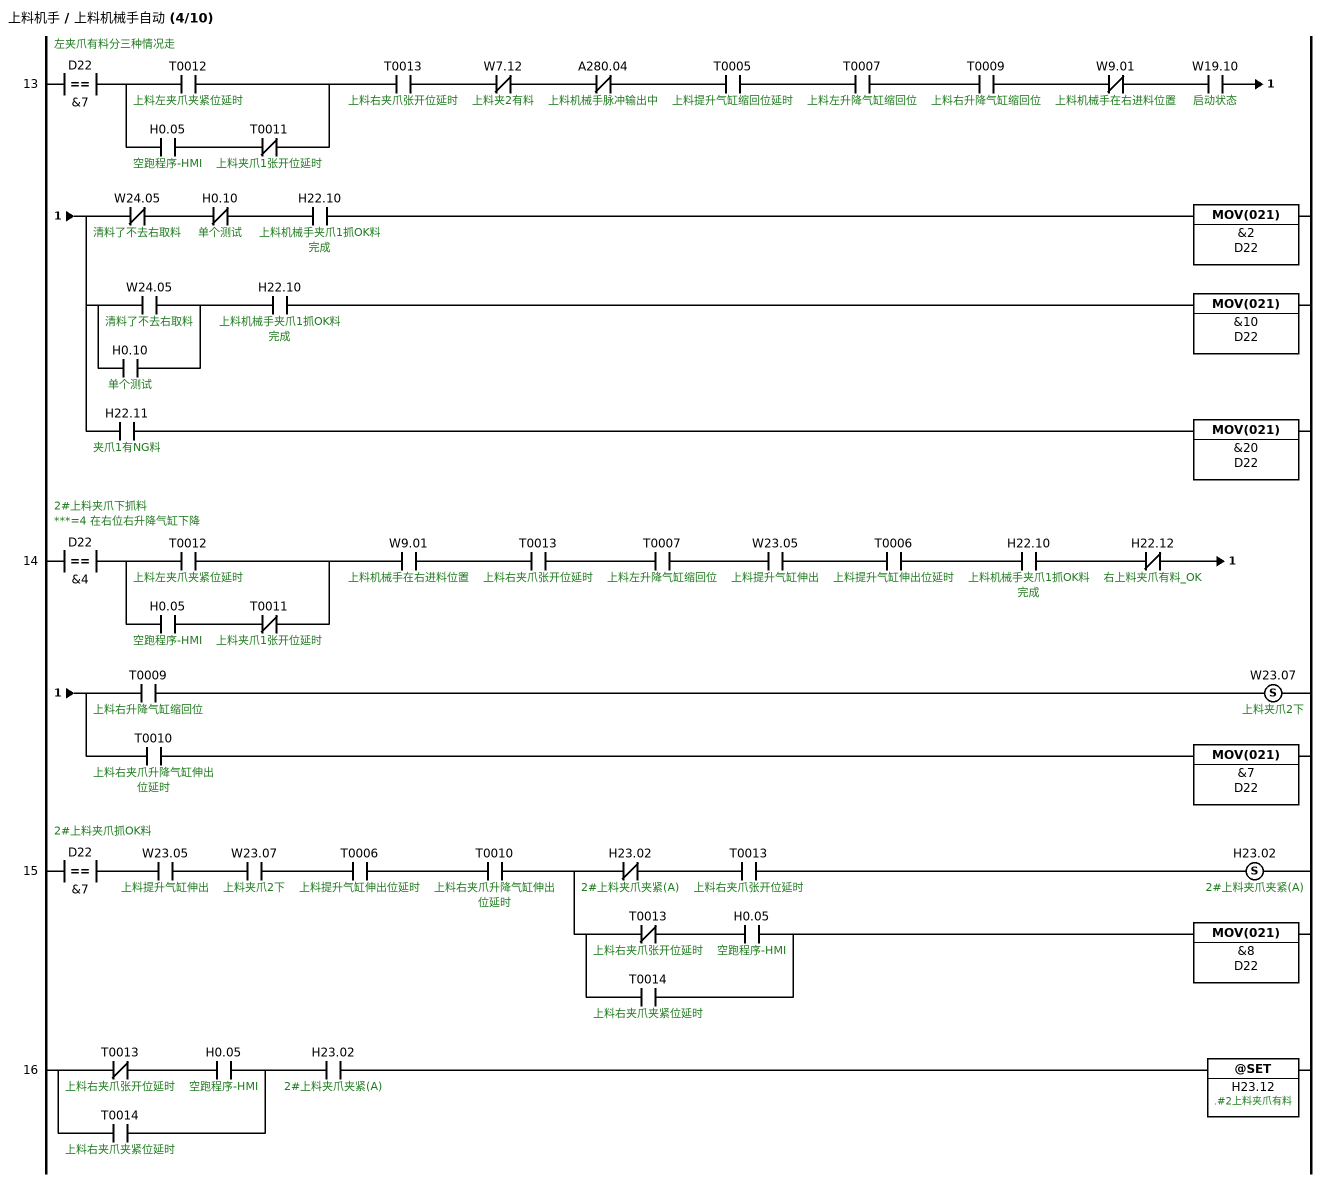
; rung 13: 左夹爪有料分三种情况走
LD=(300) D22 &7
LD T0012  ; 上料左夹爪夹紧位延时
LD H0.05  ; 空跑程序-HMI
ANDNOT T0011  ; 上料夹爪1张开位延时
ORLD
ANDLD
AND T0013  ; 上料右夹爪张开位延时
ANDNOT W7.12  ; 上料夹2有料
ANDNOT A280.04  ; 上料机械手脉冲输出中
AND T0005  ; 上料提升气缸缩回位延时
AND T0007  ; 上料左升降气缸缩回位
AND T0009  ; 上料右升降气缸缩回位
ANDNOT W9.01  ; 上料机械手在右进料位置
AND W19.10  ; 启动状态
OUT TR0
ANDNOT W24.05  ; 清料了不去右取料
ANDNOT H0.10  ; 单个测试
AND H22.10  ; 上料机械手夹爪1抓OK料完成
MOV(021) &2 D22
LD TR0
LD W24.05  ; 清料了不去右取料
OR H0.10  ; 单个测试
ANDLD
AND H22.10  ; 上料机械手夹爪1抓OK料完成
MOV(021) &10 D22
LD TR0
AND H22.11  ; 夹爪1有NG料
MOV(021) &20 D22
; rung 14: 2#上料夹爪下抓料 / ***=4 在右位右升降气缸下降
LD=(300) D22 &4
LD T0012  ; 上料左夹爪夹紧位延时
LD H0.05  ; 空跑程序-HMI
ANDNOT T0011  ; 上料夹爪1张开位延时
ORLD
ANDLD
AND W9.01  ; 上料机械手在右进料位置
AND T0013  ; 上料右夹爪张开位延时
AND T0007  ; 上料左升降气缸缩回位
AND W23.05  ; 上料提升气缸伸出
AND T0006  ; 上料提升气缸伸出位延时
AND H22.10  ; 上料机械手夹爪1抓OK料完成
ANDNOT H22.12  ; 右上料夹爪有料_OK
OUT TR0
AND T0009  ; 上料右升降气缸缩回位
SET W23.07  ; 上料夹爪2下
LD TR0
AND T0010  ; 上料右夹爪升降气缸伸出位延时
MOV(021) &7 D22
; rung 15: 2#上料夹爪抓OK料
LD=(300) D22 &7
AND W23.05  ; 上料提升气缸伸出
AND W23.07  ; 上料夹爪2下
AND T0006  ; 上料提升气缸伸出位延时
AND T0010  ; 上料右夹爪升降气缸伸出位延时
OUT TR0
ANDNOT H23.02  ; 2#上料夹爪夹紧(A)
AND T0013  ; 上料右夹爪张开位延时
SET H23.02  ; 2#上料夹爪夹紧(A)
LD TR0
LDNOT T0013  ; 上料右夹爪张开位延时
AND H0.05  ; 空跑程序-HMI
OR T0014  ; 上料右夹爪夹紧位延时
ANDLD
MOV(021) &8 D22
; rung 16
LDNOT T0013  ; 上料右夹爪张开位延时
AND H0.05  ; 空跑程序-HMI
OR T0014  ; 上料右夹爪夹紧位延时
AND H23.02  ; 2#上料夹爪夹紧(A)
@SET H23.12  ; .#2上料夹爪有料

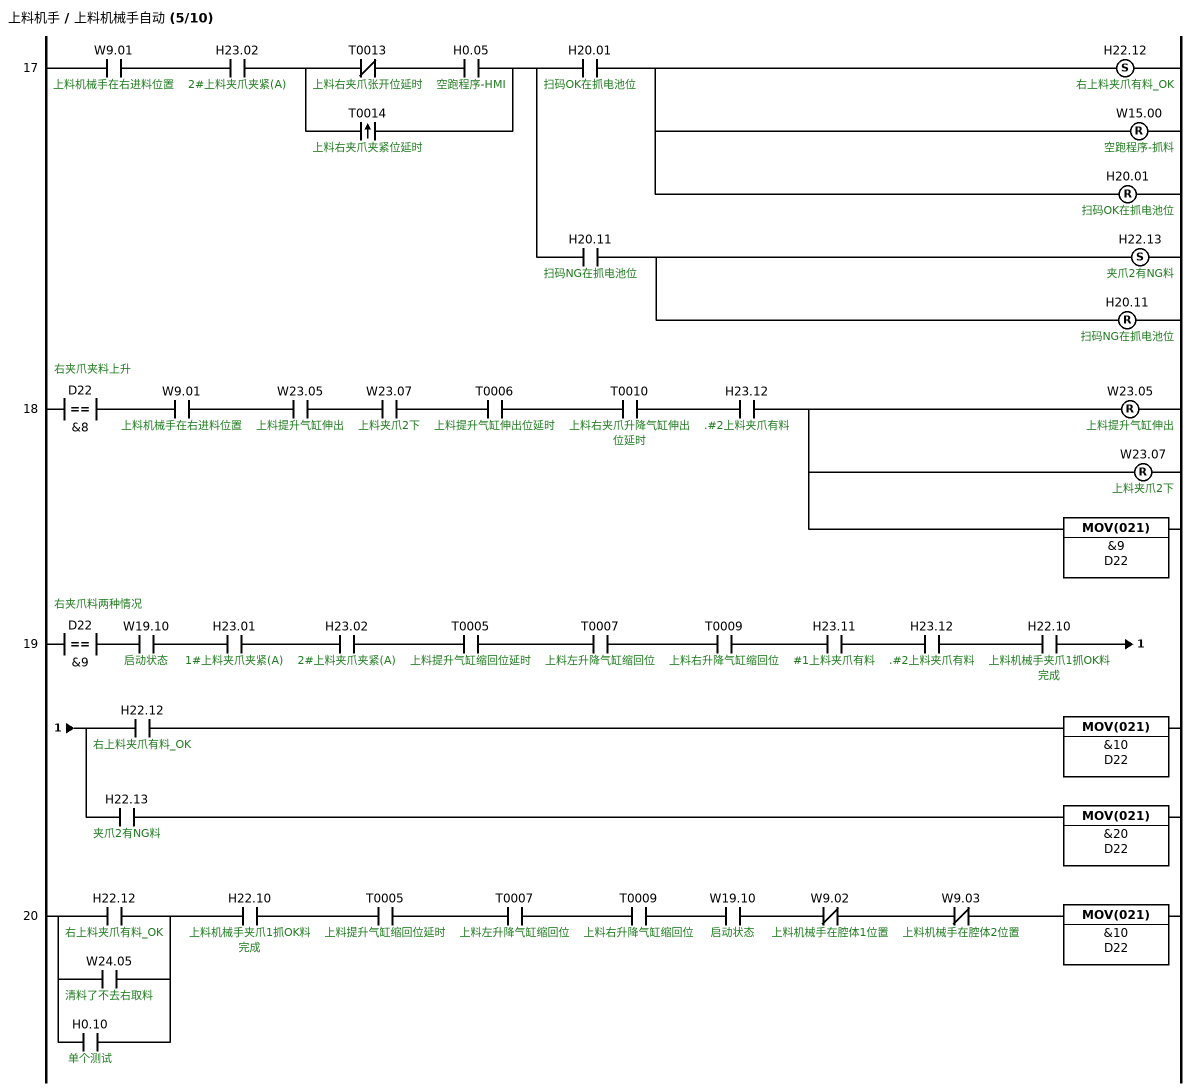
; rung 17
LD W9.01  ; 上料机械手在右进料位置
AND H23.02  ; 2#上料夹爪夹紧(A)
LDNOT T0013  ; 上料右夹爪张开位延时
AND H0.05  ; 空跑程序-HMI
@OR T0014  ; 上料右夹爪夹紧位延时
ANDLD
OUT TR0
AND H20.01  ; 扫码OK在抓电池位
SET H22.12  ; 右上料夹爪有料_OK
RSET W15.00  ; 空跑程序-抓料
RSET H20.01  ; 扫码OK在抓电池位
LD TR0
AND H20.11  ; 扫码NG在抓电池位
SET H22.13  ; 夹爪2有NG料
RSET H20.11  ; 扫码NG在抓电池位
; rung 18: 右夹爪夹料上升
LD=(300) D22 &8
AND W9.01  ; 上料机械手在右进料位置
AND W23.05  ; 上料提升气缸伸出
AND W23.07  ; 上料夹爪2下
AND T0006  ; 上料提升气缸伸出位延时
AND T0010  ; 上料右夹爪升降气缸伸出位延时
AND H23.12  ; .#2上料夹爪有料
RSET W23.05  ; 上料提升气缸伸出
RSET W23.07  ; 上料夹爪2下
MOV(021) &9 D22
; rung 19: 右夹爪料两种情况
LD=(300) D22 &9
AND W19.10  ; 启动状态
AND H23.01  ; 1#上料夹爪夹紧(A)
AND H23.02  ; 2#上料夹爪夹紧(A)
AND T0005  ; 上料提升气缸缩回位延时
AND T0007  ; 上料左升降气缸缩回位
AND T0009  ; 上料右升降气缸缩回位
AND H23.11  ; #1上料夹爪有料
AND H23.12  ; .#2上料夹爪有料
AND H22.10  ; 上料机械手夹爪1抓OK料完成
OUT TR0
AND H22.12  ; 右上料夹爪有料_OK
MOV(021) &10 D22
LD TR0
AND H22.13  ; 夹爪2有NG料
MOV(021) &20 D22
; rung 20
LD H22.12  ; 右上料夹爪有料_OK
OR W24.05  ; 清料了不去右取料
OR H0.10  ; 单个测试
AND H22.10  ; 上料机械手夹爪1抓OK料完成
AND T0005  ; 上料提升气缸缩回位延时
AND T0007  ; 上料左升降气缸缩回位
AND T0009  ; 上料右升降气缸缩回位
AND W19.10  ; 启动状态
ANDNOT W9.02  ; 上料机械手在腔体1位置
ANDNOT W9.03  ; 上料机械手在腔体2位置
MOV(021) &10 D22

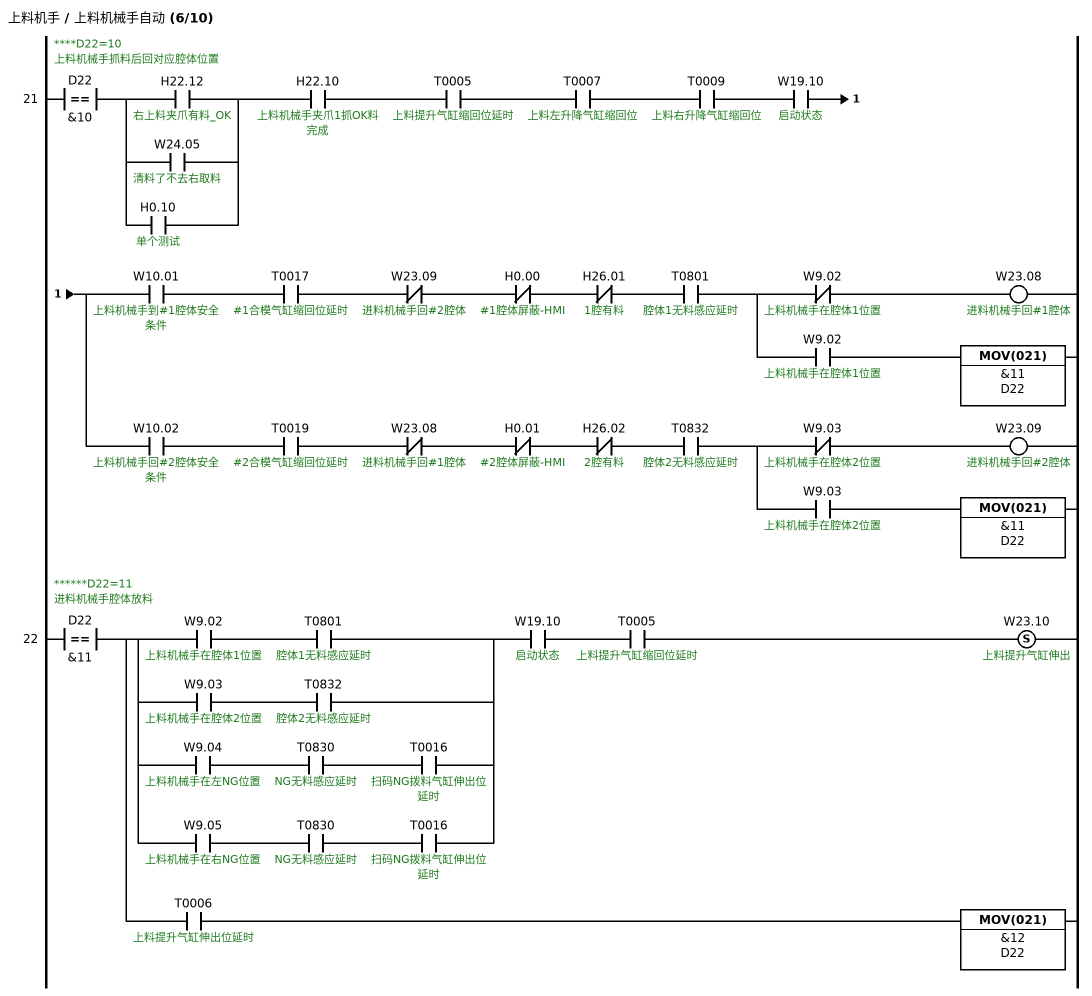
; rung 21: ****D22=10 / 上料机械手抓料后回对应腔体位置
LD=(300) D22 &10
LD H22.12  ; 右上料夹爪有料_OK
OR W24.05  ; 清料了不去右取料
OR H0.10  ; 单个测试
ANDLD
AND H22.10  ; 上料机械手夹爪1抓OK料完成
AND T0005  ; 上料提升气缸缩回位延时
AND T0007  ; 上料左升降气缸缩回位
AND T0009  ; 上料右升降气缸缩回位
AND W19.10  ; 启动状态
OUT TR0
AND W10.01  ; 上料机械手到#1腔体安全条件
AND T0017  ; #1合模气缸缩回位延时
ANDNOT W23.09  ; 进料机械手回#2腔体
ANDNOT H0.00  ; #1腔体屏蔽-HMI
ANDNOT H26.01  ; 1腔有料
AND T0801  ; 腔体1无料感应延时
OUT TR1
ANDNOT W9.02  ; 上料机械手在腔体1位置
OUT W23.08  ; 进料机械手回#1腔体
LD TR1
AND W9.02  ; 上料机械手在腔体1位置
MOV(021) &11 D22
LD TR0
AND W10.02  ; 上料机械手回#2腔体安全条件
AND T0019  ; #2合模气缸缩回位延时
ANDNOT W23.08  ; 进料机械手回#1腔体
ANDNOT H0.01  ; #2腔体屏蔽-HMI
ANDNOT H26.02  ; 2腔有料
AND T0832  ; 腔体2无料感应延时
OUT TR0
ANDNOT W9.03  ; 上料机械手在腔体2位置
OUT W23.09  ; 进料机械手回#2腔体
LD TR0
AND W9.03  ; 上料机械手在腔体2位置
MOV(021) &11 D22
; rung 22: ******D22=11 / 进料机械手腔体放料
LD=(300) D22 &11
OUT TR0
LD W9.02  ; 上料机械手在腔体1位置
AND T0801  ; 腔体1无料感应延时
LD W9.03  ; 上料机械手在腔体2位置
AND T0832  ; 腔体2无料感应延时
ORLD
LD W9.04  ; 上料机械手在左NG位置
AND T0830  ; NG无料感应延时
AND T0016  ; 扫码NG拨料气缸伸出位延时
ORLD
LD W9.05  ; 上料机械手在右NG位置
AND T0830  ; NG无料感应延时
AND T0016  ; 扫码NG拨料气缸伸出位延时
ORLD
ANDLD
AND W19.10  ; 启动状态
AND T0005  ; 上料提升气缸缩回位延时
SET W23.10  ; 上料提升气缸伸出
LD TR0
AND T0006  ; 上料提升气缸伸出位延时
MOV(021) &12 D22

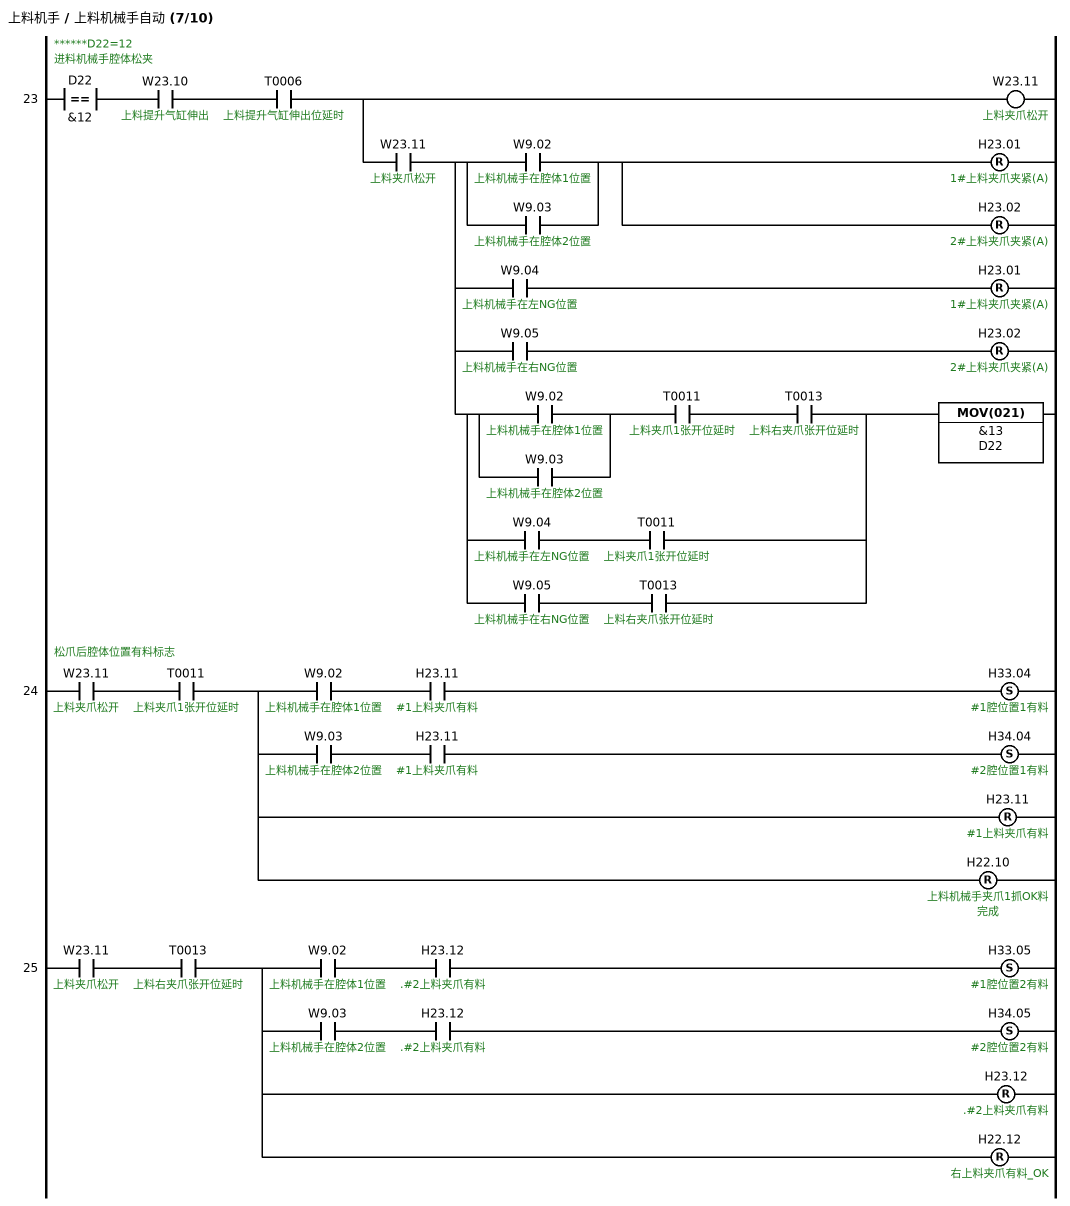
; rung 23: ******D22=12 / 进料机械手腔体松夹
LD=(300) D22 &12
AND W23.10  ; 上料提升气缸伸出
AND T0006  ; 上料提升气缸伸出位延时
OUT W23.11  ; 上料夹爪松开
AND W23.11  ; 上料夹爪松开
OUT TR0
LD W9.02  ; 上料机械手在腔体1位置
OR W9.03  ; 上料机械手在腔体2位置
ANDLD
RSET H23.01  ; 1#上料夹爪夹紧(A)
RSET H23.02  ; 2#上料夹爪夹紧(A)
LD TR0
AND W9.04  ; 上料机械手在左NG位置
RSET H23.01  ; 1#上料夹爪夹紧(A)
LD TR0
AND W9.05  ; 上料机械手在右NG位置
RSET H23.02  ; 2#上料夹爪夹紧(A)
LD TR0
LD W9.02  ; 上料机械手在腔体1位置
OR W9.03  ; 上料机械手在腔体2位置
AND T0011  ; 上料夹爪1张开位延时
AND T0013  ; 上料右夹爪张开位延时
LD W9.04  ; 上料机械手在左NG位置
AND T0011  ; 上料夹爪1张开位延时
ORLD
LD W9.05  ; 上料机械手在右NG位置
AND T0013  ; 上料右夹爪张开位延时
ORLD
ANDLD
MOV(021) &13 D22
; rung 24: 松爪后腔体位置有料标志
LD W23.11  ; 上料夹爪松开
AND T0011  ; 上料夹爪1张开位延时
OUT TR0
AND W9.02  ; 上料机械手在腔体1位置
AND H23.11  ; #1上料夹爪有料
SET H33.04  ; #1腔位置1有料
LD TR0
AND W9.03  ; 上料机械手在腔体2位置
AND H23.11  ; #1上料夹爪有料
SET H34.04  ; #2腔位置1有料
LD TR0
RSET H23.11  ; #1上料夹爪有料
RSET H22.10  ; 上料机械手夹爪1抓OK料完成
; rung 25
LD W23.11  ; 上料夹爪松开
AND T0013  ; 上料右夹爪张开位延时
OUT TR0
AND W9.02  ; 上料机械手在腔体1位置
AND H23.12  ; .#2上料夹爪有料
SET H33.05  ; #1腔位置2有料
LD TR0
AND W9.03  ; 上料机械手在腔体2位置
AND H23.12  ; .#2上料夹爪有料
SET H34.05  ; #2腔位置2有料
LD TR0
RSET H23.12  ; .#2上料夹爪有料
RSET H22.12  ; 右上料夹爪有料_OK

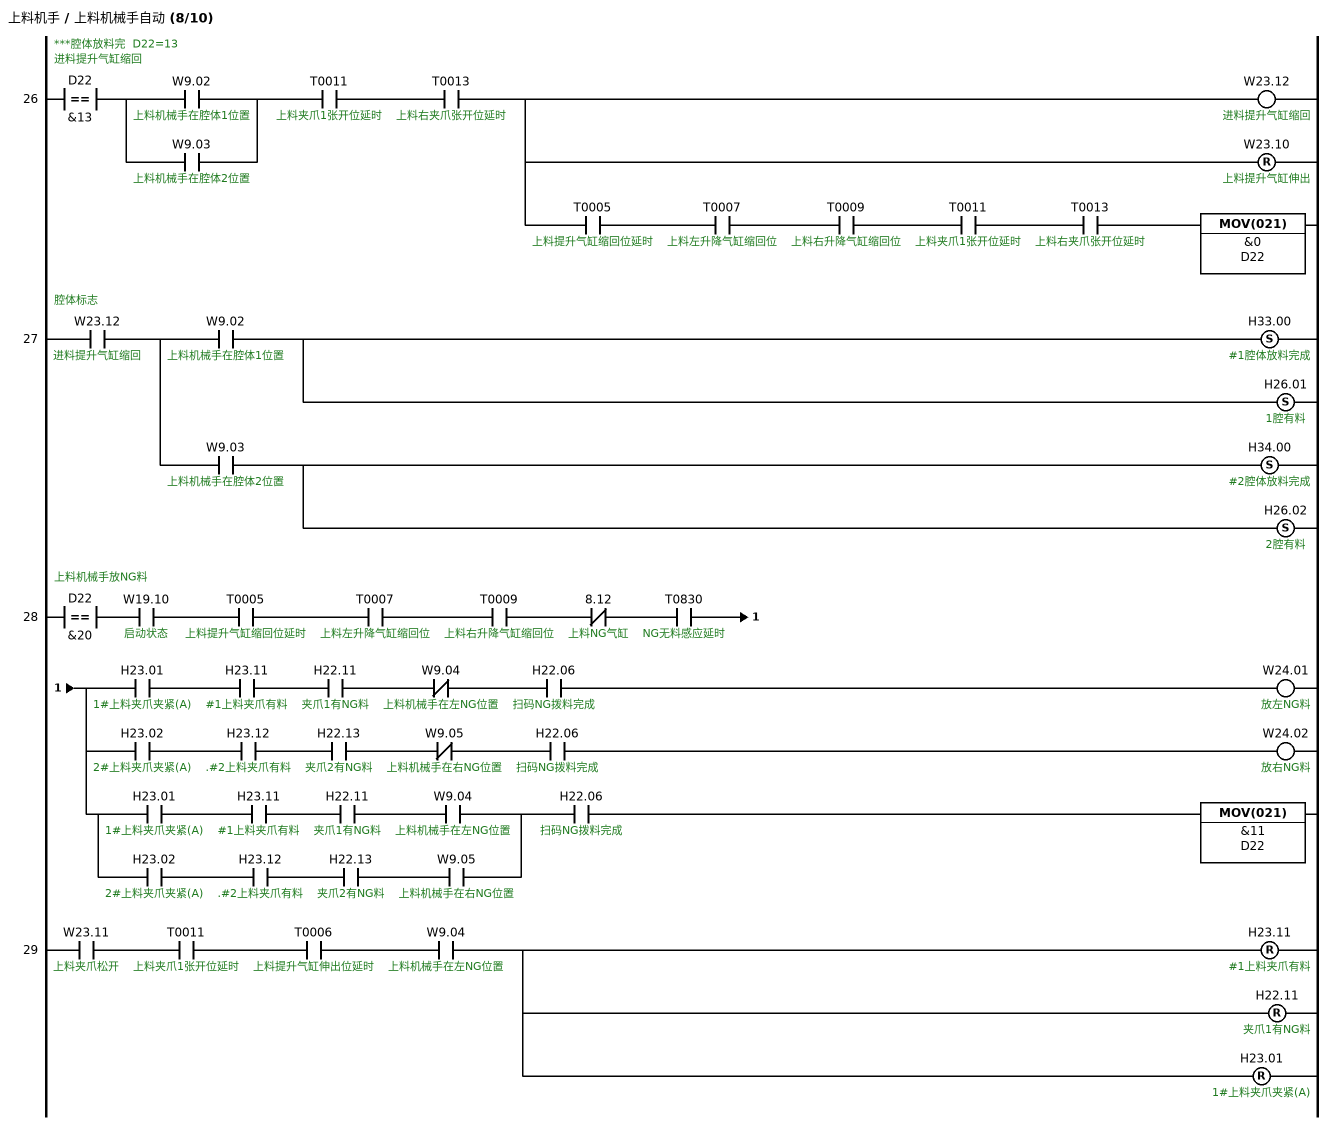
; rung 26: ***腔体放料完  D22=13 / 进料提升气缸缩回
LD=(300) D22 &13
LD W9.02  ; 上料机械手在腔体1位置
OR W9.03  ; 上料机械手在腔体2位置
ANDLD
AND T0011  ; 上料夹爪1张开位延时
AND T0013  ; 上料右夹爪张开位延时
OUT W23.12  ; 进料提升气缸缩回
RSET W23.10  ; 上料提升气缸伸出
AND T0005  ; 上料提升气缸缩回位延时
AND T0007  ; 上料左升降气缸缩回位
AND T0009  ; 上料右升降气缸缩回位
AND T0011  ; 上料夹爪1张开位延时
AND T0013  ; 上料右夹爪张开位延时
MOV(021) &0 D22
; rung 27: 腔体标志
LD W23.12  ; 进料提升气缸缩回
OUT TR0
AND W9.02  ; 上料机械手在腔体1位置
SET H33.00  ; #1腔体放料完成
SET H26.01  ; 1腔有料
LD TR0
AND W9.03  ; 上料机械手在腔体2位置
SET H34.00  ; #2腔体放料完成
SET H26.02  ; 2腔有料
; rung 28: 上料机械手放NG料
LD=(300) D22 &20
AND W19.10  ; 启动状态
AND T0005  ; 上料提升气缸缩回位延时
AND T0007  ; 上料左升降气缸缩回位
AND T0009  ; 上料右升降气缸缩回位
ANDNOT 8.12  ; 上料NG气缸
AND T0830  ; NG无料感应延时
OUT TR0
AND H23.01  ; 1#上料夹爪夹紧(A)
AND H23.11  ; #1上料夹爪有料
AND H22.11  ; 夹爪1有NG料
ANDNOT W9.04  ; 上料机械手在左NG位置
AND H22.06  ; 扫码NG拨料完成
OUT W24.01  ; 放左NG料
LD TR0
AND H23.02  ; 2#上料夹爪夹紧(A)
AND H23.12  ; .#2上料夹爪有料
AND H22.13  ; 夹爪2有NG料
ANDNOT W9.05  ; 上料机械手在右NG位置
AND H22.06  ; 扫码NG拨料完成
OUT W24.02  ; 放右NG料
LD TR0
LD H23.01  ; 1#上料夹爪夹紧(A)
AND H23.11  ; #1上料夹爪有料
AND H22.11  ; 夹爪1有NG料
AND W9.04  ; 上料机械手在左NG位置
LD H23.02  ; 2#上料夹爪夹紧(A)
AND H23.12  ; .#2上料夹爪有料
AND H22.13  ; 夹爪2有NG料
AND W9.05  ; 上料机械手在右NG位置
ORLD
ANDLD
AND H22.06  ; 扫码NG拨料完成
MOV(021) &11 D22
; rung 29
LD W23.11  ; 上料夹爪松开
AND T0011  ; 上料夹爪1张开位延时
AND T0006  ; 上料提升气缸伸出位延时
AND W9.04  ; 上料机械手在左NG位置
RSET H23.11  ; #1上料夹爪有料
RSET H22.11  ; 夹爪1有NG料
RSET H23.01  ; 1#上料夹爪夹紧(A)

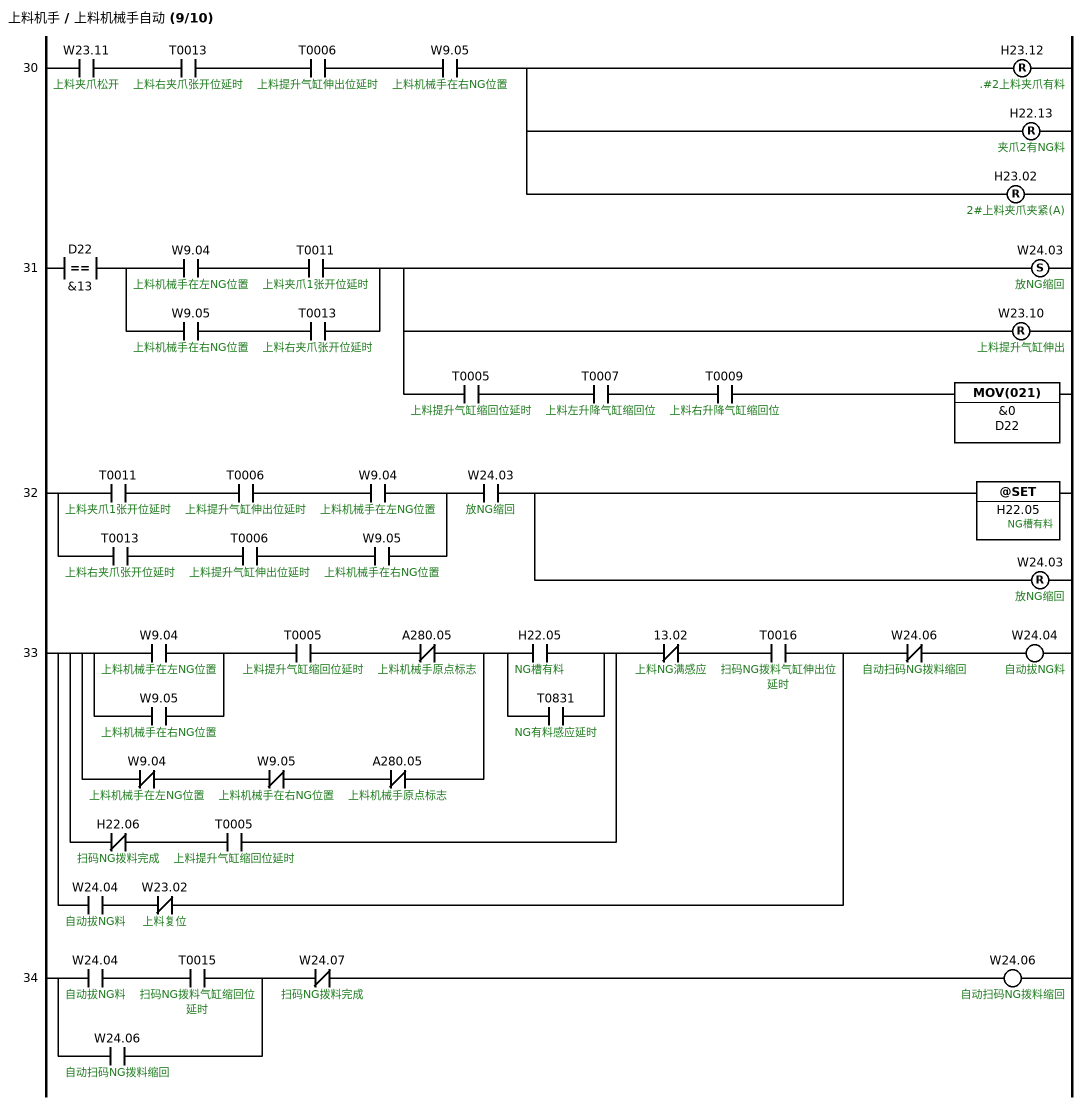
; rung 30
LD W23.11  ; 上料夹爪松开
AND T0013  ; 上料右夹爪张开位延时
AND T0006  ; 上料提升气缸伸出位延时
AND W9.05  ; 上料机械手在右NG位置
RSET H23.12  ; .#2上料夹爪有料
RSET H22.13  ; 夹爪2有NG料
RSET H23.02  ; 2#上料夹爪夹紧(A)
; rung 31
LD=(300) D22 &13
LD W9.04  ; 上料机械手在左NG位置
AND T0011  ; 上料夹爪1张开位延时
LD W9.05  ; 上料机械手在右NG位置
AND T0013  ; 上料右夹爪张开位延时
ORLD
ANDLD
SET W24.03  ; 放NG缩回
RSET W23.10  ; 上料提升气缸伸出
AND T0005  ; 上料提升气缸缩回位延时
AND T0007  ; 上料左升降气缸缩回位
AND T0009  ; 上料右升降气缸缩回位
MOV(021) &0 D22
; rung 32
LD T0011  ; 上料夹爪1张开位延时
AND T0006  ; 上料提升气缸伸出位延时
AND W9.04  ; 上料机械手在左NG位置
LD T0013  ; 上料右夹爪张开位延时
AND T0006  ; 上料提升气缸伸出位延时
AND W9.05  ; 上料机械手在右NG位置
ORLD
AND W24.03  ; 放NG缩回
@SET H22.05  ; NG槽有料
RSET W24.03  ; 放NG缩回
; rung 33
LD W9.04  ; 上料机械手在左NG位置
OR W9.05  ; 上料机械手在右NG位置
AND T0005  ; 上料提升气缸缩回位延时
ANDNOT A280.05  ; 上料机械手原点标志
LDNOT W9.04  ; 上料机械手在左NG位置
ANDNOT W9.05  ; 上料机械手在右NG位置
ANDNOT A280.05  ; 上料机械手原点标志
ORLD
LD H22.05  ; NG槽有料
OR T0831  ; NG有料感应延时
ANDLD
LDNOT H22.06  ; 扫码NG拨料完成
AND T0005  ; 上料提升气缸缩回位延时
ORLD
ANDNOT 13.02  ; 上料NG满感应
AND T0016  ; 扫码NG拨料气缸伸出位延时
LD W24.04  ; 自动拔NG料
ANDNOT W23.02  ; 上料复位
ORLD
ANDNOT W24.06  ; 自动扫码NG拨料缩回
OUT W24.04  ; 自动拔NG料
; rung 34
LD W24.04  ; 自动拔NG料
AND T0015  ; 扫码NG拨料气缸缩回位延时
OR W24.06  ; 自动扫码NG拨料缩回
ANDNOT W24.07  ; 扫码NG拨料完成
OUT W24.06  ; 自动扫码NG拨料缩回

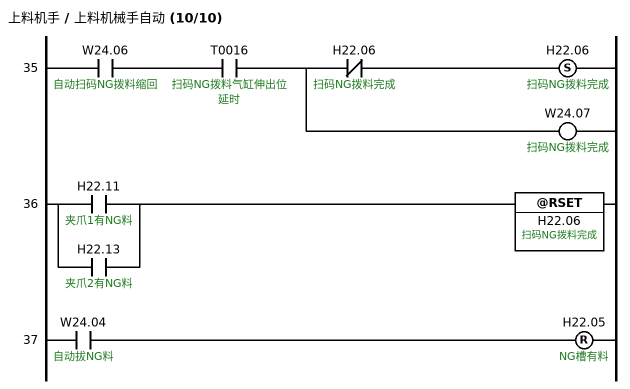
; rung 35
LD W24.06  ; 自动扫码NG拨料缩回
AND T0016  ; 扫码NG拨料气缸伸出位延时
OUT TR0
ANDNOT H22.06  ; 扫码NG拨料完成
SET H22.06  ; 扫码NG拨料完成
LD TR0
OUT W24.07  ; 扫码NG拨料完成
; rung 36
LD H22.11  ; 夹爪1有NG料
OR H22.13  ; 夹爪2有NG料
@RSET H22.06  ; 扫码NG拨料完成
; rung 37
LD W24.04  ; 自动拔NG料
RSET H22.05  ; NG槽有料

### Section 伺服参数

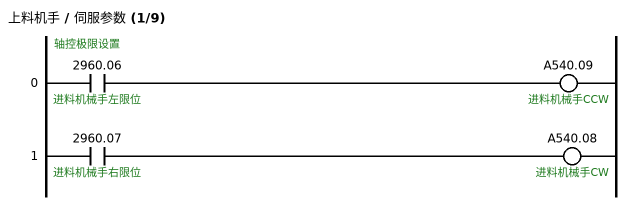
; rung 0: 轴控极限设置
LD 2960.06  ; 进料机械手左限位
OUT A540.09  ; 进料机械手CCW
; rung 1
LD 2960.07  ; 进料机械手右限位
OUT A540.08  ; 进料机械手CW

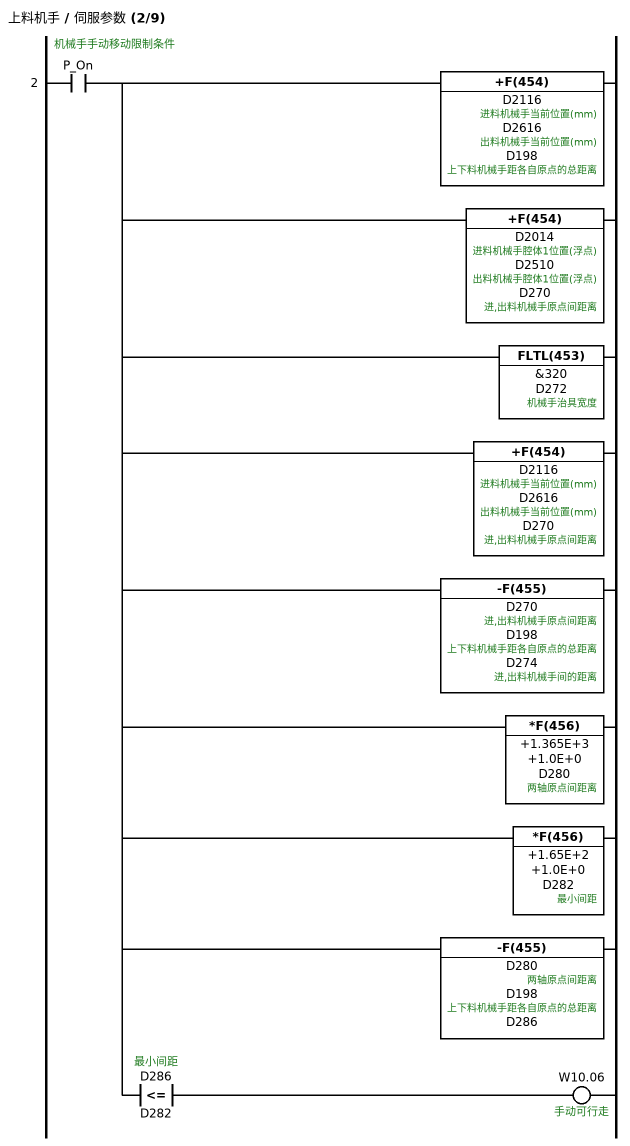
; rung 2: 机械手手动移动限制条件
LD P_On
+F(454) D2116 D2616 D198  ; 进料机械手当前位置(mm), 出料机械手当前位置(mm), 上下料机械手距各自原点的总距离
+F(454) D2014 D2510 D270  ; 进料机械手腔体1位置(浮点), 出料机械手腔体1位置(浮点), 进,出料机械手原点间距离
FLTL(453) &320 D272  ; 机械手治具宽度
+F(454) D2116 D2616 D270  ; 进料机械手当前位置(mm), 出料机械手当前位置(mm), 进,出料机械手原点间距离
-F(455) D270 D198 D274  ; 进,出料机械手原点间距离, 上下料机械手距各自原点的总距离, 进,出料机械手间的距离
*F(456) +1.365E+3 +1.0E+0 D280  ; 两轴原点间距离
*F(456) +1.65E+2 +1.0E+0 D282  ; 最小间距
-F(455) D280 D198 D286  ; 两轴原点间距离, 上下料机械手距各自原点的总距离
AND<=F(332) D286 D282  ; 最小间距
OUT W10.06  ; 手动可行走

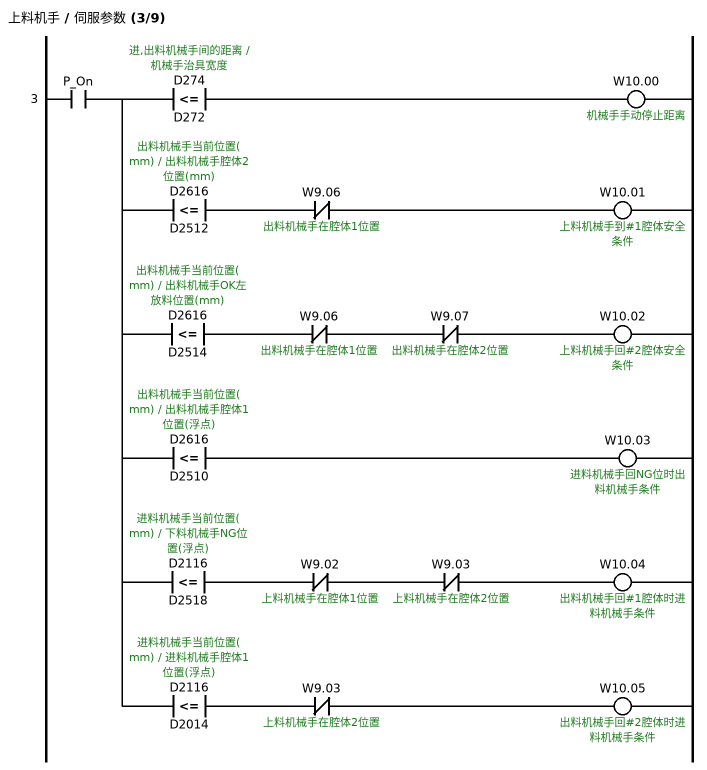
; rung 3
LD P_On
OUT TR0
AND<=(315) D274 D272  ; 进,出料机械手间的距离, 机械手治具宽度
OUT W10.00  ; 机械手手动停止距离
LD TR0
AND<=(315) D2616 D2512  ; 出料机械手当前位置(mm), 出料机械手腔体2位置(mm)
ANDNOT W9.06  ; 出料机械手在腔体1位置
OUT W10.01  ; 上料机械手到#1腔体安全条件
LD TR0
AND<=(315) D2616 D2514  ; 出料机械手当前位置(mm), 出料机械手OK左放料位置(mm)
ANDNOT W9.06  ; 出料机械手在腔体1位置
ANDNOT W9.07  ; 出料机械手在腔体2位置
OUT W10.02  ; 上料机械手回#2腔体安全条件
LD TR0
AND<=(315) D2616 D2510  ; 出料机械手当前位置(mm), 出料机械手腔体1位置(浮点)
OUT W10.03  ; 进料机械手回NG位时出料机械手条件
LD TR0
AND<=(315) D2116 D2518  ; 进料机械手当前位置(mm), 下料机械手NG位置(浮点)
ANDNOT W9.02  ; 上料机械手在腔体1位置
ANDNOT W9.03  ; 上料机械手在腔体2位置
OUT W10.04  ; 出料机械手回#1腔体时进料机械手条件
LD TR0
AND<=(315) D2116 D2014  ; 进料机械手当前位置(mm), 进料机械手腔体1位置(浮点)
ANDNOT W9.03  ; 上料机械手在腔体2位置
OUT W10.05  ; 出料机械手回#2腔体时进料机械手条件

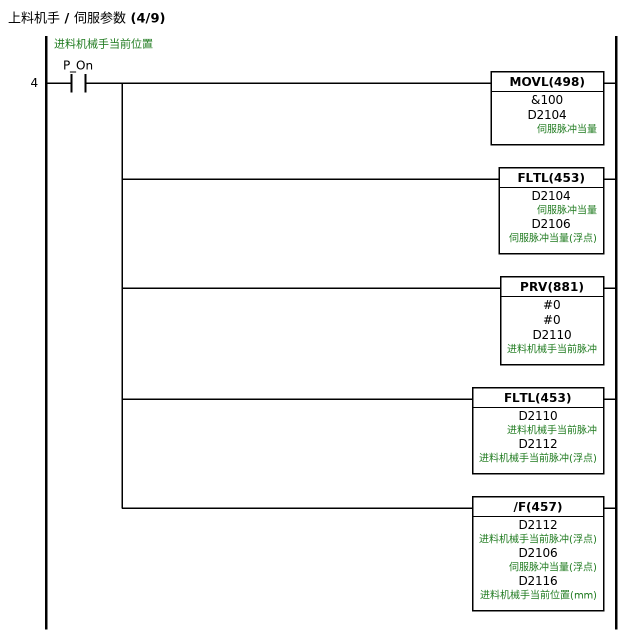
; rung 4: 进料机械手当前位置
LD P_On
MOVL(498) &100 D2104  ; 伺服脉冲当量
FLTL(453) D2104 D2106  ; 伺服脉冲当量, 伺服脉冲当量(浮点)
PRV(881) #0 #0 D2110  ; 进料机械手当前脉冲
FLTL(453) D2110 D2112  ; 进料机械手当前脉冲, 进料机械手当前脉冲(浮点)
/F(457) D2112 D2106 D2116  ; 进料机械手当前脉冲(浮点), 伺服脉冲当量(浮点), 进料机械手当前位置(mm)

